(* Logix 5000 project; controller Arrow3 vendor 1 type 14 code 235 rev 36.11; software revision 36.00 *)

TASK MainTask (continuous, watchdog 500 ms) : MainProgram
TASK SafetyTask (periodic, rate 20 ms, priority 10, watchdog 20 ms, safety) : SafetyProgram

MODULES
   Local : vendor 1 type 14 code 235 (5069 0, rev 36.11)
      VRQx : vendor 1609 type 7 code 1234 (Ethernet 192.168.1.10, rev 1.4, StandardDataDriven RPI 20 ms)
END_MODULES

TYPE STR_20 :
STRUCT
   DATA : SINT[20];
END_STRUCT
END_TYPE

PROGRAM MainProgram   (* main routine MainRoutine *)
VAR
   b : BOOL := 1;
   DI1_4_INPUTTYPE_GET : MESSAGE;
        MessageParameters(ServiceCode := 16#000e, DestinationTag := DI1_4_INPUTTYPE_GET_VAL, ...)
   DI1_4_INPUTTYPE_GET_VAL : UINT;
   DI1_4_INPUTTYPE_SET : MESSAGE;
        MessageParameters(ServiceCode := 16#0010, LocalElement := DI1_4_INPUTTYPE_SET_VAL, ...)
   DI1_4_INPUTTYPE_SET_VAL : UINT;
   DI1_4_INPUTTYPE_TRG_GET : BOOL;
   DI1_4_INPUTTYPE_TRG_SET : BOOL;
   DI1_8_FORCEENABLE_GET : MESSAGE;
        MessageParameters(ServiceCode := 16#000e, DestinationTag := DI1_8_FORCEENABLE_GET_VAL, ...)
   DI1_8_FORCEENABLE_GET_VAL : UINT;
   DI1_8_FORCEENABLE_SET : MESSAGE;
        MessageParameters(ServiceCode := 16#0010, LocalElement := DI1_8_FORCEENABLE_SET_VAL, ...)
   DI1_8_FORCEENABLE_SET_VAL : UINT;
   DI1_8_FORCEENABLE_TRG_GET : BOOL;
   DI1_8_FORCEENABLE_TRG_SET : BOOL;
   DI1_8_FORCESTATE_GET : MESSAGE;
        MessageParameters(ServiceCode := 16#000e, DestinationTag := DI1_8_FORCESTATE_GET_VAL, ...)
   DI1_8_FORCESTATE_GET_VAL : UINT;
   DI1_8_FORCESTATE_SET : MESSAGE;
        MessageParameters(ServiceCode := 16#0010, LocalElement := DI1_8_FORCESTATE_SET_VAL, ...)
   DI1_8_FORCESTATE_SET_VAL : UINT;
   DI1_8_FORCESTATE_TRG_GET : BOOL;
   DI1_8_FORCESTATE_TRG_SET : BOOL;
   DI1_8_LOGICINVERT_GET : MESSAGE;
        MessageParameters(ServiceCode := 16#000e, DestinationTag := DI1_8_LOGICINVERT_GET_VAL, ...)
   DI1_8_LOGICINVERT_GET_VAL : UINT;
   DI1_8_LOGICINVERT_SET : MESSAGE;
        MessageParameters(ServiceCode := 16#0010, LocalElement := DI1_8_LOGICINVERT_SET_VAL, ...)
   DI1_8_LOGICINVERT_SET_VAL : UINT;
   DI1_8_LOGICINVERT_TRG_GET : BOOL;
   DI1_8_LOGICINVERT_TRG_SET : BOOL;
   DI1_CHNLERRSTS_GET : MESSAGE;
        MessageParameters(ServiceCode := 16#000e, DestinationTag := DI1_CHNLERRSTS_GET_VAL, ...)
   DI1_CHNLERRSTS_GET_VAL : UINT;
   DI1_CHNLERRSTS_TRG_GET : BOOL;
   DI1_DEBOUNCEDUR_GET : MESSAGE;
        MessageParameters(ServiceCode := 16#000e, DestinationTag := DI1_DEBOUNCEDUR_GET_VAL, ...)
   DI1_DEBOUNCEDUR_GET_VAL : UINT;
   DI1_DEBOUNCEDUR_SET : MESSAGE;
        MessageParameters(ServiceCode := 16#0010, LocalElement := DI1_DEBOUNCEDUR_SET_VAL, ...)
   DI1_DEBOUNCEDUR_SET_VAL : UINT;
   DI1_DEBOUNCEDUR_TRG_GET : BOOL := 1;
   DI1_DEBOUNCEDUR_TRG_SET : BOOL;
   DI1_HOLDDUR_SET : MESSAGE;
        MessageParameters(ServiceCode := 16#0010, LocalElement := DI1_HOLDDUR_SET_VAL, ...)
   DI1_HOLDDUR_SET_VAL : UINT;
   DI1_HOLDDUR_TRG_SET : BOOL;
   DI2_CHNLERRSTS_GET : MESSAGE;
        MessageParameters(ServiceCode := 16#000e, DestinationTag := DI2_CHNLERRSTS_GET_VAL, ...)
   DI2_CHNLERRSTS_GET_VAL : UINT;
   DI2_CHNLERRSTS_TRG_GET : BOOL;
   DI2_DEBOUNCEDUR_GET : MESSAGE;
        MessageParameters(ServiceCode := 16#000e, DestinationTag := DI2_DEBOUNCEDUR_GET_VAL, ...)
   DI2_DEBOUNCEDUR_GET_VAL : UINT;
   DI2_DEBOUNCEDUR_SET : MESSAGE;
        MessageParameters(ServiceCode := 16#0010, LocalElement := DI2_DEBOUNCEDUR_SET_VAL, ...)
   DI2_DEBOUNCEDUR_SET_VAL : UINT;
   DI2_DEBOUNCEDUR_TRG_GET : BOOL := 1;
   DI2_DEBOUNCEDUR_TRG_SET : BOOL;
   DI2_HOLDDUR_SET : MESSAGE;
        MessageParameters(ServiceCode := 16#0010, LocalElement := DI2_HOLDDUR_SET_VAL, ...)
   DI2_HOLDDUR_SET_VAL : UINT;
   DI2_HOLDDUR_TRG_SET : BOOL;
   DI3_CHNLERRSTS_GET : MESSAGE;
        MessageParameters(ServiceCode := 16#000e, DestinationTag := DI3_CHNLERRSTS_GET_VAL, ...)
   DI3_CHNLERRSTS_GET_VAL : UINT;
   DI3_CHNLERRSTS_TRG_GET : BOOL;
   DI3_DEBOUNCEDUR_GET : MESSAGE;
        MessageParameters(ServiceCode := 16#000e, DestinationTag := DI3_DEBOUNCEDUR_GET_VAL, ...)
   DI3_DEBOUNCEDUR_GET_VAL : UINT;
   DI3_DEBOUNCEDUR_SET : MESSAGE;
        MessageParameters(ServiceCode := 16#0010, LocalElement := DI3_DEBOUNCEDUR_SET_VAL, ...)
   DI3_DEBOUNCEDUR_SET_VAL : UINT;
   DI3_DEBOUNCEDUR_TRG_GET : BOOL := 1;
   DI3_DEBOUNCEDUR_TRG_SET : BOOL;
   DI3_HOLDDUR_SET : MESSAGE;
        MessageParameters(ServiceCode := 16#0010, LocalElement := DI3_HOLDDUR_SET_VAL, ...)
   DI3_HOLDDUR_SET_VAL : DINT;
   DI3_HOLDDUR_TRG_SET : BOOL;
   DI4_CHNLERRSTS_GET : MESSAGE;
        MessageParameters(ServiceCode := 16#000e, DestinationTag := DI4_CHNLERRSTS_GET_VAL, ...)
   DI4_CHNLERRSTS_GET_VAL : UINT;
   DI4_CHNLERRSTS_TRG_GET : BOOL;
   DI4_DEBOUNCEDUR_GET : MESSAGE;
        MessageParameters(ServiceCode := 16#000e, DestinationTag := DI4_DEBOUNCEDUR_GET_VAL, ...)
   DI4_DEBOUNCEDUR_GET_VAL : UINT;
   DI4_DEBOUNCEDUR_SET : MESSAGE;
        MessageParameters(ServiceCode := 16#0010, LocalElement := DI4_DEBOUNCEDUR_SET_VAL, ...)
   DI4_DEBOUNCEDUR_SET_VAL : UINT;
   DI4_DEBOUNCEDUR_TRG_GET : BOOL := 1;
   DI4_DEBOUNCEDUR_TRG_SET : BOOL;
   DI4_HOLDDUR_SET : MESSAGE;
        MessageParameters(ServiceCode := 16#0010, LocalElement := DI4_HOLDDUR_SET_VAL, ...)
   DI4_HOLDDUR_SET_VAL : UINT;
   DI4_HOLDDUR_TRG_SET : BOOL;
   DI5_8_INPUTTYPE_GET : MESSAGE;
        MessageParameters(ServiceCode := 16#000e, DestinationTag := DI5_8_INPUTTYPE_GET_VAL, ...)
   DI5_8_INPUTTYPE_GET_VAL : UINT;
   DI5_8_INPUTTYPE_SET : MESSAGE;
        MessageParameters(ServiceCode := 16#0010, LocalElement := DI5_8_INPUTTYPE_SET_VAL, ...)
   DI5_8_INPUTTYPE_SET_VAL : UINT;
   DI5_8_INPUTTYPE_TRG_GET : BOOL;
   DI5_8_INPUTTYPE_TRG_SET : BOOL;
   DI5_CHNLERRSTS_GET : MESSAGE;
        MessageParameters(ServiceCode := 16#000e, DestinationTag := DI5_CHNLERRSTS_GET_VAL, ...)
   DI5_CHNLERRSTS_GET_VAL : UINT;
   DI5_CHNLERRSTS_TRG_GET : BOOL;
   DI5_DEBOUNCEDUR_GET : MESSAGE;
        MessageParameters(ServiceCode := 16#000e, DestinationTag := DI5_DEBOUNCEDUR_GET_VAL, ...)
   DI5_DEBOUNCEDUR_GET_VAL : UINT;
   DI5_DEBOUNCEDUR_SET : MESSAGE;
        MessageParameters(ServiceCode := 16#0010, LocalElement := DI5_DEBOUNCEDUR_SET_VAL, ...)
   DI5_DEBOUNCEDUR_SET_VAL : UINT;
   DI5_DEBOUNCEDUR_TRG_GET : BOOL;
   DI5_DEBOUNCEDUR_TRG_SET : BOOL;
   DI5_HOLDDUR_SET : MESSAGE;
        MessageParameters(ServiceCode := 16#0010, LocalElement := DI5_HOLDDUR_SET_VAL, ...)
   DI5_HOLDDUR_SET_VAL : UINT;
   DI5_HOLDDUR_TRG_SET : BOOL;
   DI6_CHNLERRSTS_GET : MESSAGE;
        MessageParameters(ServiceCode := 16#000e, DestinationTag := DI6_CHNLERRSTS_GET_VAL, ...)
   DI6_CHNLERRSTS_GET_VAL : UINT;
   DI6_CHNLERRSTS_TRG_GET : BOOL;
   DI6_DEBOUNCEDUR_GET : MESSAGE;
        MessageParameters(ServiceCode := 16#000e, DestinationTag := DI6_DEBOUNCEDUR_GET_VAL, ...)
   DI6_DEBOUNCEDUR_GET_VAL : UINT;
   DI6_DEBOUNCEDUR_SET : MESSAGE;
        MessageParameters(ServiceCode := 16#0010, LocalElement := DI6_DEBOUNCEDUR_SET_VAL, ...)
   DI6_DEBOUNCEDUR_SET_VAL : UINT;
   DI6_DEBOUNCEDUR_TRG_GET : BOOL;
   DI6_DEBOUNCEDUR_TRG_SET : BOOL;
   DI6_HOLDDUR_SET : MESSAGE;
        MessageParameters(ServiceCode := 16#0010, LocalElement := DI6_HOLDDUR_SET_VAL, ...)
   DI6_HOLDDUR_SET_VAL : UINT;
   DI6_HOLDDUR_TRG_SET : BOOL;
   DI7_CHNLERRSTS_GET : MESSAGE;
        MessageParameters(ServiceCode := 16#000e, DestinationTag := DI7_CHNLERRSTS_GET_VAL, ...)
   DI7_CHNLERRSTS_GET_VAL : UINT;
   DI7_CHNLERRSTS_TRG_GET : BOOL;
   DI7_DEBOUNCEDUR_GET : MESSAGE;
        MessageParameters(ServiceCode := 16#000e, DestinationTag := DI7_DEBOUNCEDUR_GET_VAL, ...)
   DI7_DEBOUNCEDUR_GET_VAL : UINT;
   DI7_DEBOUNCEDUR_SET : MESSAGE;
        MessageParameters(ServiceCode := 16#0010, LocalElement := DI7_DEBOUNCEDUR_SET_VAL, ...)
   DI7_DEBOUNCEDUR_SET_VAL : UINT;
   DI7_DEBOUNCEDUR_TRG_GET : BOOL;
   DI7_DEBOUNCEDUR_TRG_SET : BOOL;
   DI7_HOLDDUR_SET : MESSAGE;
        MessageParameters(ServiceCode := 16#0010, LocalElement := DI7_HOLDDUR_SET_VAL, ...)
   DI7_HOLDDUR_SET_VAL : UINT;
   DI7_HOLDDUR_TRG_SET : BOOL;
   DI8_CHNLERRSTS_GET : MESSAGE;
        MessageParameters(ServiceCode := 16#000e, DestinationTag := DI8_CHNLERRSTS_GET_VAL, ...)
   DI8_CHNLERRSTS_GET_VAL : UINT;
   DI8_CHNLERRSTS_TRG_GET : BOOL;
   DI8_DEBOUNCEDUR_GET : MESSAGE;
        MessageParameters(ServiceCode := 16#000e, DestinationTag := DI8_DEBOUNCEDUR_GET_VAL, ...)
   DI8_DEBOUNCEDUR_GET_VAL : UINT;
   DI8_DEBOUNCEDUR_SET : MESSAGE;
        MessageParameters(ServiceCode := 16#0010, LocalElement := DI7_DEBOUNCEDUR_SET_VAL, ...)
   DI8_DEBOUNCEDUR_SET_VAL : UINT;
   DI8_DEBOUNCEDUR_TRG_GET : BOOL;
   DI8_DEBOUNCEDUR_TRG_SET : BOOL;
   DI8_HOLDDUR_SET : MESSAGE;
        MessageParameters(ServiceCode := 16#0010, LocalElement := DI8_HOLDDUR_SET_VAL, ...)
   DI8_HOLDDUR_SET_VAL : UINT;
   DI8_HOLDDUR_TRG_SET : BOOL;
   DI_BOTHEDGE_INT_GET : MESSAGE;
        MessageParameters(ServiceCode := 16#000e, DestinationTag := DI_BOTHEDGE_INT_GET_VAL, ...)
   DI_BOTHEDGE_INT_GET_VAL : UINT;
   DI_BOTHEDGE_INT_SET : MESSAGE;
        MessageParameters(ServiceCode := 16#0010, LocalElement := DI_BOTHEDGE_INT_SET_VAL, ...)
   DI_BOTHEDGE_INT_SET_VAL : DINT;
   DI_BOTHEDGE_INT_TRG_GET : BOOL;
   DI_BOTHEDGE_INT_TRG_SET : BOOL;
   DI_HITOLOEDGE_INT_GET : MESSAGE;
        MessageParameters(ServiceCode := 16#000e, DestinationTag := DI_HITOLOEDGE_INT_GET_VAL, ...)
   DI_HITOLOEDGE_INT_GET_VAL : UINT;
   DI_HITOLOEDGE_INT_SET : MESSAGE;
        MessageParameters(ServiceCode := 16#0010, LocalElement := DI_HITOLOEDGE_INT_SET_VAL, ...)
   DI_HITOLOEDGE_INT_SET_VAL : DINT;
   DI_HITOLOEDGE_INT_TRG_GET : BOOL;
   DI_HITOLOEDGE_INT_TRG_SET : BOOL;
   DI_LOTOHIEDGE_INT_GET : MESSAGE;
        MessageParameters(ServiceCode := 16#000e, DestinationTag := DI_LOTOHIEDGE_INT_GET_VAL, ...)
   DI_LOTOHIEDGE_INT_GET_VAL : UINT;
   DI_LOTOHIEDGE_INT_SET : MESSAGE;
        MessageParameters(ServiceCode := 16#0010, LocalElement := DI_LOTOHIEDGE_INT_SET_VAL, ...)
   DI_LOTOHIEDGE_INT_SET_VAL : DINT;
   DI_LOTOHIEDGE_INT_TRG_GET : BOOL;
   DI_LOTOHIEDGE_INT_TRG_SET : BOOL;
   DIO_CHNLPOS_ERRSTATUS_GET : MESSAGE;
        MessageParameters(ServiceCode := 16#000e, DestinationTag := DIO_CHNLPOS_ERRSTATUS_GET_VAL, ...)
   DIO_CHNLPOS_ERRSTATUS_GET_VAL : UINT;
   DIO_CHNLPOS_ERRSTATUS_TRG_GET : BOOL;
   DIO_FAULTRECOVERYENABLE_GET : MESSAGE;
        MessageParameters(ServiceCode := 16#000e, DestinationTag := DIO_FAULTRECOVERYENABLE_GET_VAL, ...)
   DIO_FAULTRECOVERYENABLE_GET_VAL : UINT;
   DIO_FAULTRECOVERYENABLE_SET : MESSAGE;
        MessageParameters(ServiceCode := 16#0010, LocalElement := DIO_FAULTRECOVERYENABLE_SET_VAL, ...)
   DIO_FAULTRECOVERYENABLE_SET_VAL : UINT;
   DIO_FAULTRECOVERYENABLE_TRG_GET : BOOL;
   DIO_FAULTRECOVERYENABLE_TRG_SET : BOOL;
   DIO_IDENT_DEVICEID_GET : MESSAGE;
        MessageParameters(ServiceCode := 16#000e, DestinationTag := DIO_IDENT_DEVICEID_GET_VAL, ...)
   DIO_IDENT_DEVICEID_GET_VAL : UDINT;
   DIO_IDENT_DEVICEID_TRG_GET : BOOL;
   DIO_IDENT_DEVICENAME_GET : MESSAGE;
        MessageParameters(ServiceCode := 16#000e, DestinationTag := DIO_IDENT_DEVICENAME_GET_VAL, ...)
   DIO_IDENT_DEVICENAME_GET_VAL : STR_20;
   DIO_IDENT_DEVICENAME_TRG_GET : BOOL;
   DIO_IDENT_DEVICETYPE_GET : MESSAGE;
        MessageParameters(ServiceCode := 16#000e, DestinationTag := DIO_IDENT_DEVICETYPE_GET_VAL, ...)
   DIO_IDENT_DEVICETYPE_GET_VAL : UDINT;
   DIO_IDENT_DEVICETYPE_TRG_GET : BOOL;
   DIO_IDENT_HWREV_GET : MESSAGE;
        MessageParameters(ServiceCode := 16#000e, DestinationTag := DIO_IDENT_HWREV_GET_VAL, ...)
   DIO_IDENT_HWREV_GET_VAL : STR_20;
   DIO_IDENT_HWREV_TRG_GET : BOOL;
   DIO_IDENT_SERIALNO_GET : MESSAGE;
        MessageParameters(ServiceCode := 16#000e, DestinationTag := DIO_IDENT_SERIALNO_GET_VAL, ...)
   DIO_IDENT_SERIALNO_GET_VAL : STR_20;
   DIO_IDENT_SERIALNO_TRG_GET : BOOL;
   DIO_IDENT_SWPARTNO_GET : MESSAGE;
        MessageParameters(ServiceCode := 16#000e, DestinationTag := DIO_IDENT_SWPARTNO_GET_VAL, ...)
   DIO_IDENT_SWPARTNO_GET_VAL : STR_20;
   DIO_IDENT_SWPARTNO_TRG_GET : BOOL;
   DIO_IDENT_SWREV_GET : MESSAGE;
        MessageParameters(ServiceCode := 16#000e, DestinationTag := DIO_IDENT_SWREV_GET_VAL, ...)
   DIO_IDENT_SWREV_GET_VAL : STR_20;
   DIO_IDENT_SWREV_TRG_GET : BOOL;
   DIO_IDENT_VARIANTID_GET : MESSAGE;
        MessageParameters(ServiceCode := 16#000e, DestinationTag := DIO_IDENT_VARIANTID_GET_VAL, ...)
   DIO_IDENT_VARIANTID_GET_VAL : STR_20;
   DIO_IDENT_VARIANTID_TRG_GET : BOOL;
   DIO_IDENT_VENDORID_GET : MESSAGE;
        MessageParameters(ServiceCode := 16#000e, DestinationTag := DIO_IDENT_VENDORID_GET_VAL, ...)
   DIO_IDENT_VENDORID_GET_VAL : UDINT;
   DIO_IDENT_VENDORID_TRG_GET : BOOL;
   DIO_IDENT_VENDORNAME_GET : MESSAGE;
        MessageParameters(ServiceCode := 16#000e, DestinationTag := DIO_IDENT_VENDORNAME_GET_VAL, ...)
   DIO_IDENT_VENDORNAME_GET_VAL : STR_20;
   DIO_IDENT_VENDORNAME_TRG_GET : BOOL;
   DIO_MEMORYLIFECYCLE_GET : MESSAGE;
        MessageParameters(ServiceCode := 16#000e, DestinationTag := DIO_MEMORYLIFECYCLE_GET_VAL, ...)
   DIO_MEMORYLIFECYCLE_GET_VAL : UDINT;
   DIO_MEMORYLIFECYCLE_TRG_GET : BOOL;
   DIO_OPERATIONTIME_HR_GET : MESSAGE;
        MessageParameters(ServiceCode := 16#000e, DestinationTag := DIO_OPERATIONTIME_HR_GET_VAL, ...)
   DIO_OPERATIONTIME_HR_GET_VAL : UDINT;
   DIO_OPERATIONTIME_HR_TRG_GET : BOOL;
   DIO_OPERATIONTIME_MIN_GET : MESSAGE;
        MessageParameters(ServiceCode := 16#000e, DestinationTag := DIO_OPERATIONTIME_MIN_GET_VAL, ...)
   DIO_OPERATIONTIME_MIN_GET_VAL : UDINT;
   DIO_OPERATIONTIME_MIN_TRG_GET : BOOL;
   DO1_8_BUSFAULTENABLE_GET : MESSAGE;
        MessageParameters(ServiceCode := 16#000e, DestinationTag := DO1_8_BUSFAULTENABLE_GET_VAL, ...)
   DO1_8_BUSFAULTENABLE_GET_VAL : UINT;
   DO1_8_BUSFAULTENABLE_SET : MESSAGE;
        MessageParameters(ServiceCode := 16#0010, LocalElement := DO1_8_BUSFAULTENABLE_SET_VAL, ...)
   DO1_8_BUSFAULTENABLE_SET_VAL : UINT;
   DO1_8_BUSFAULTENABLE_TRG_GET : BOOL;
   DO1_8_BUSFAULTENABLE_TRG_SET : BOOL;
   DO1_8_BUSFAULTSTATE_GET : MESSAGE;
        MessageParameters(ServiceCode := 16#000e, DestinationTag := DO1_8_BUSFAULTSTATE_GET_VAL, ...)
   DO1_8_BUSFAULTSTATE_GET_VAL : UINT;
   DO1_8_BUSFAULTSTATE_SET : MESSAGE;
        MessageParameters(ServiceCode := 16#0010, LocalElement := DO1_8_BUSFAULTSTATE_SET_VAL, ...)
   DO1_8_BUSFAULTSTATE_SET_VAL : UINT;
   DO1_8_BUSFAULTSTATE_TRG_GET : BOOL;
   DO1_8_BUSFAULTSTATE_TRG_SET : BOOL;
   DO1_8_FORCEENABLE_GET : MESSAGE;
        MessageParameters(ServiceCode := 16#000e, DestinationTag := DO1_8_FORCEENABLE_GET_VAL, ...)
   DO1_8_FORCEENABLE_GET_VAL : UINT;
   DO1_8_FORCEENABLE_SET : MESSAGE;
        MessageParameters(ServiceCode := 16#0010, LocalElement := DO1_8_FORCEENABLE_SET_VAL, ...)
   DO1_8_FORCEENABLE_SET_VAL : UINT;
   DO1_8_FORCEENABLE_TRG_GET : BOOL;
   DO1_8_FORCEENABLE_TRG_SET : BOOL;
   DO1_8_FORCESTATE_GET : MESSAGE;
        MessageParameters(ServiceCode := 16#000e, DestinationTag := DO1_8_FORCESTATE_GET_VAL, ...)
   DO1_8_FORCESTATE_GET_VAL : UINT;
   DO1_8_FORCESTATE_SET : MESSAGE;
        MessageParameters(ServiceCode := 16#0010, LocalElement := DO1_8_FORCESTATE_SET_VAL, ...)
   DO1_8_FORCESTATE_SET_VAL : UINT;
   DO1_8_FORCESTATE_TRG_GET : BOOL;
   DO1_8_FORCESTATE_TRG_SET : BOOL;
   DO1_8_IDLEMODEENABLE_GET : MESSAGE;
        MessageParameters(ServiceCode := 16#000e, DestinationTag := DO1_8_IDLEMODEENABLE_GET_VAL, ...)
   DO1_8_IDLEMODEENABLE_GET_VAL : UINT;
   DO1_8_IDLEMODEENABLE_SET : MESSAGE;
        MessageParameters(ServiceCode := 16#0010, LocalElement := DO1_8_IDLEMODEENABLE_SET_VAL, ...)
   DO1_8_IDLEMODEENABLE_SET_VAL : UINT;
   DO1_8_IDLEMODEENABLE_TRG_GET : BOOL;
   DO1_8_IDLEMODEENABLE_TRG_SET : BOOL;
   DO1_8_IDLEMODESTATE_GET : MESSAGE;
        MessageParameters(ServiceCode := 16#000e, DestinationTag := DO1_8_IDLEMODESTATE_GET_VAL, ...)
   DO1_8_IDLEMODESTATE_GET_VAL : UINT;
   DO1_8_IDLEMODESTATE_SET : MESSAGE;
        MessageParameters(ServiceCode := 16#0010, LocalElement := DO1_8_IDLEMODESTATE_SET_VAL, ...)
   DO1_8_IDLEMODESTATE_SET_VAL : UINT;
   DO1_8_IDLEMODESTATE_TRG_GET : BOOL;
   DO1_8_IDLEMODESTATE_TRG_SET : BOOL;
   DO1_CHNLERRSTS_GET : MESSAGE;
        MessageParameters(ServiceCode := 16#000e, DestinationTag := DO1_CHNLERRSTS_GET_VAL, ...)
   DO1_CHNLERRSTS_GET_VAL : UINT;
   DO1_CHNLERRSTS_TRG_GET : BOOL;
   DO2_CHNLERRSTS_GET : MESSAGE;
        MessageParameters(ServiceCode := 16#000e, DestinationTag := DO2_CHNLERRSTS_GET_VAL, ...)
   DO2_CHNLERRSTS_GET_VAL : UINT;
   DO2_CHNLERRSTS_TRG_GET : BOOL;
   DO3_CHNLERRSTS_GET : MESSAGE;
        MessageParameters(ServiceCode := 16#000e, DestinationTag := DO3_CHNLERRSTS_GET_VAL, ...)
   DO3_CHNLERRSTS_GET_VAL : UINT;
   DO3_CHNLERRSTS_TRG_GET : BOOL;
   DO4_CHNLERRSTS_GET : MESSAGE;
        MessageParameters(ServiceCode := 16#000e, DestinationTag := DO4_CHNLERRSTS_GET_VAL, ...)
   DO4_CHNLERRSTS_GET_VAL : UINT;
   DO4_CHNLERRSTS_TRG_GET : BOOL;
   DO5_CHNLERRSTS_GET : MESSAGE;
        MessageParameters(ServiceCode := 16#000e, DestinationTag := DO5_CHNLERRSTS_GET_VAL, ...)
   DO5_CHNLERRSTS_GET_VAL : UINT;
   DO5_CHNLERRSTS_TRG_GET : BOOL;
   DO6_CHNLERRSTS_GET : MESSAGE;
        MessageParameters(ServiceCode := 16#000e, DestinationTag := DO6_CHNLERRSTS_GET_VAL, ...)
   DO6_CHNLERRSTS_GET_VAL : UINT;
   DO6_CHNLERRSTS_TRG_GET : BOOL;
   DO7_CHNLERRSTS_GET : MESSAGE;
        MessageParameters(ServiceCode := 16#000e, DestinationTag := DO7_CHNLERRSTS_GET_VAL, ...)
   DO7_CHNLERRSTS_GET_VAL : UINT;
   DO7_CHNLERRSTS_TRG_GET : BOOL;
   DO8_CHNLERRSTS_GET : MESSAGE;
        MessageParameters(ServiceCode := 16#000e, DestinationTag := DO8_CHNLERRSTS_GET_VAL, ...)
   DO8_CHNLERRSTS_GET_VAL : UINT;
   DO8_CHNLERRSTS_TRG_GET : BOOL;
   DO_IDLEMODEENABLE_GET : MESSAGE;
        MessageParameters(ServiceCode := 16#000e, DestinationTag := DO_IDLEMODEENABLE_GET_VAL, ...)
   DO_IDLEMODEENABLE_GET_VAL : UINT;
   DO_IDLEMODEENABLE_SET : MESSAGE;
        MessageParameters(ServiceCode := 16#0010, LocalElement := DO_IDLEMODEENABLE_SET_VAL, ...)
   DO_IDLEMODEENABLE_SET_VAL : UINT;
   DO_IDLEMODEENABLE_TRG_GET : BOOL;
   DO_IDLEMODEENABLE_TRG_SET : BOOL;
   ENABLE_IMPLICIT_SET : MESSAGE;
        MessageParameters(ServiceCode := 16#0010, LocalElement := ENABLE_IMPLICIT_SET_CMD_VAL, ...)
   ENABLE_IMPLICIT_SET_CMD_VAL : UINT;
   ENABLE_IMPLICIT_TRG_SET : BOOL;
   ISEM_BCKPLANE_IDENT_DEVICEID_GET : MESSAGE;
        MessageParameters(ServiceCode := 16#000e, DestinationTag := ISEM_BCKPLANE_IDENT_DEVICEID_GET_VAL, ...)
   ISEM_BCKPLANE_IDENT_DEVICEID_GET_VAL : UDINT;
   ISEM_BCKPLANE_IDENT_DEVICEID_TRG_GET : BOOL;
   ISEM_BCKPLANE_IDENT_DEVICENAME_GET : MESSAGE;
        MessageParameters(ServiceCode := 16#000e, DestinationTag := ISEM_BCKPLANE_IDENT_DEVICENAME_GET_VAL, ...)
   ISEM_BCKPLANE_IDENT_DEVICENAME_GET_VAL : STR_20;
   ISEM_BCKPLANE_IDENT_DEVICENAME_TRG_GET : BOOL;
   ISEM_BCKPLANE_IDENT_DEVICETYPE_GET : MESSAGE;
        MessageParameters(ServiceCode := 16#000e, DestinationTag := ISEM_BCKPLANE_IDENT_DEVICETYPE_GET_VAL, ...)
   ISEM_BCKPLANE_IDENT_DEVICETYPE_GET_VAL : UDINT;
   ISEM_BCKPLANE_IDENT_DEVICETYPE_TRG_GET : BOOL;
   ISEM_BCKPLANE_IDENT_HWREV_GET : MESSAGE;
        MessageParameters(ServiceCode := 16#000e, DestinationTag := ISEM_BCKPLANE_IDENT_HWREV_GET_VAL, ...)
   ISEM_BCKPLANE_IDENT_HWREV_GET_VAL : STR_20;
   ISEM_BCKPLANE_IDENT_HWREV_TRG_GET : BOOL;
   ISEM_BCKPLANE_IDENT_SERIALNO_GET : MESSAGE;
        MessageParameters(ServiceCode := 16#000e, DestinationTag := ISEM_BCKPLANE_IDENT_SERIALNO_GET_VAL, ...)
   ISEM_BCKPLANE_IDENT_SERIALNO_GET_VAL : STR_20;
   ISEM_BCKPLANE_IDENT_SERIALNO_TRG_GET : BOOL;
   ISEM_BCKPLANE_IDENT_SWPARTNO_GET : MESSAGE;
        MessageParameters(ServiceCode := 16#000e, DestinationTag := ISEM_BCKPLANE_IDENT_SWPARTNO_GET_VAL, ...)
   ISEM_BCKPLANE_IDENT_SWPARTNO_GET_VAL : STR_20;
   ISEM_BCKPLANE_IDENT_SWPARTNO_TRG_GET : BOOL;
   ISEM_BCKPLANE_IDENT_SWREV_GET : MESSAGE;
        MessageParameters(ServiceCode := 16#000e, DestinationTag := ISEM_BCKPLANE_IDENT_SWREV_GET_VAL, ...)
   ISEM_BCKPLANE_IDENT_SWREV_GET_VAL : STR_20;
   ISEM_BCKPLANE_IDENT_SWREV_TRG_GET : BOOL;
   ISEM_BCKPLANE_IDENT_VARIANTID_GET : MESSAGE;
        MessageParameters(ServiceCode := 16#000e, DestinationTag := ISEM_BCKPLANE_IDENT_VARIANTID_GET_VAL, ...)
   ISEM_BCKPLANE_IDENT_VARIANTID_GET_VAL : STR_20;
   ISEM_BCKPLANE_IDENT_VARIANTID_TRG_GET : BOOL;
   ISEM_BCKPLANE_IDENT_VENDORID_GET : MESSAGE;
        MessageParameters(ServiceCode := 16#000e, DestinationTag := ISEM_BCKPLANE_IDENT_VENDORID_GET_VAL, ...)
   ISEM_BCKPLANE_IDENT_VENDORID_GET_VAL : UDINT;
   ISEM_BCKPLANE_IDENT_VENDORID_TRG_GET : BOOL;
   ISEM_BCKPLANE_IDENT_VENDORNAME_GET : MESSAGE;
        MessageParameters(ServiceCode := 16#000e, DestinationTag := ISEM_BCKPLANE_IDENT_VENDORNAME_GET_VAL, ...)
   ISEM_BCKPLANE_IDENT_VENDORNAME_GET_VAL : STR_20;
   ISEM_BCKPLANE_IDENT_VENDORNAME_TRG_GET : BOOL;
   ISEMDIAG_ApplPresHysteresis_GET : MESSAGE;
        MessageParameters(ServiceCode := 16#000e, DestinationTag := ISEMDIAG_ApplPresHysteresis_Get_VAL, ...)
   ISEMDIAG_ApplPresHysteresis_Get_VAL : INT;
   ISEMDIAG_ApplPresHysteresis_SET : MESSAGE;
        MessageParameters(ServiceCode := 16#0010, LocalElement := ISEMDIAG_ApplPresHysteresis_Set_VAL, ...)
   ISEMDIAG_ApplPresHysteresis_Set_VAL : INT;
   ISEMDIAG_ApplPresHysteresis_TRG_GET : BOOL;
   ISEMDIAG_ApplPresHysteresis_TRG_SET : BOOL;
   ISEMDIAG_FAULTEVNTBITS_GET : MESSAGE;
        MessageParameters(ServiceCode := 16#000e, DestinationTag := ISEMDIAG_FAULTEVNTBITS_GET_VAL, ...)
   ISEMDIAG_FAULTEVNTBITS_GET_VAL : UDINT;
   ISEMDIAG_FAULTEVNTBITS_TRG_GET : BOOL;
   ISEMDIAG_FAULTEVNTCOUNT_GET : MESSAGE;
        MessageParameters(ServiceCode := 16#000e, DestinationTag := ISEMDIAG_FAULTEVNTCOUNT_GET_VAL, ...)
   ISEMDIAG_FAULTEVNTCOUNT_GET_VAL : UINT;
   ISEMDIAG_FAULTEVNTCOUNT_TRG_GET : BOOL;
   ISEMDIAG_IDENT_DEVICEID_GET : MESSAGE;
        MessageParameters(ServiceCode := 16#000e, DestinationTag := ISEMDIAG_IDENT_DEVICEID_GET_VAL, ...)
   ISEMDIAG_IDENT_DEVICEID_GET_VAL : UDINT;
   ISEMDIAG_IDENT_DEVICEID_TRG_GET : BOOL;
   ISEMDIAG_IDENT_DEVICENAME_GET : MESSAGE;
        MessageParameters(ServiceCode := 16#000e, DestinationTag := ISEMDIAG_IDENT_DEVICENAME_GET_VAL, ...)
   ISEMDIAG_IDENT_DEVICENAME_GET_VAL : STR_20;
   ISEMDIAG_IDENT_DEVICENAME_TRG_GET : BOOL;
   ISEMDIAG_IDENT_DEVICETYPE_GET : MESSAGE;
        MessageParameters(ServiceCode := 16#000e, DestinationTag := ISEMDIAG_IDENT_DEVICETYPE_GET_VAL, ...)
   ISEMDIAG_IDENT_DEVICETYPE_GET_VAL : UDINT;
   ISEMDIAG_IDENT_DEVICETYPE_TRG_GET : BOOL;
   ISEMDIAG_IDENT_HWREV_GET : MESSAGE;
        MessageParameters(ServiceCode := 16#000e, DestinationTag := ISEMDIAG_IDENT_HWREV_GET_VAL, ...)
   ISEMDIAG_IDENT_HWREV_GET_VAL : STR_20;
   ISEMDIAG_IDENT_HWREV_TRG_GET : BOOL;
   ISEMDIAG_IDENT_SERIALNO_GET : MESSAGE;
        MessageParameters(ServiceCode := 16#000e, DestinationTag := ISEMDIAG_IDENT_SERIALNO_GET_VAL, ...)
   ISEMDIAG_IDENT_SERIALNO_GET_VAL : STR_20;
   ISEMDIAG_IDENT_SERIALNO_TRG_GET : BOOL;
   ISEMDIAG_IDENT_SWPARTNO_GET : MESSAGE;
        MessageParameters(ServiceCode := 16#000e, DestinationTag := ISEMDIAG_IDENT_SWPARTNO_GET_VAL, ...)
   ISEMDIAG_IDENT_SWPARTNO_GET_VAL : STR_20;
   ISEMDIAG_IDENT_SWPARTNO_TRG_GET : BOOL;
   ISEMDIAG_IDENT_SWREV_GET : MESSAGE;
        MessageParameters(ServiceCode := 16#000e, DestinationTag := ISEMDIAG_IDENT_SWREV_GET_VAL, ...)
   ISEMDIAG_IDENT_SWREV_GET_VAL : STR_20;
   ISEMDIAG_IDENT_SWREV_TRG_GET : BOOL;
   ISEMDIAG_IDENT_VARIANTID_GET : MESSAGE;
        MessageParameters(ServiceCode := 16#000e, DestinationTag := ISEMDIAG_IDENT_VARIANTID_GET_VAL, ...)
   ISEMDIAG_IDENT_VARIANTID_GET_VAL : STR_20;
   ISEMDIAG_IDENT_VARIANTID_TRG_GET : BOOL;
   ISEMDIAG_IDENT_VENDORID_GET : MESSAGE;
        MessageParameters(ServiceCode := 16#000e, DestinationTag := ISEMDIAG_IDENT_VENDORID_GET_VAL, ...)
   ISEMDIAG_IDENT_VENDORID_GET_VAL : UDINT;
   ISEMDIAG_IDENT_VENDORID_TRG_GET : BOOL;
   ISEMDIAG_IDENT_VENDORNAME_GET : MESSAGE;
        MessageParameters(ServiceCode := 16#000e, DestinationTag := ISEMDIAG_IDENT_VENDORNAME_GET_VAL, ...)
   ISEMDIAG_IDENT_VENDORNAME_GET_VAL : STR_20;
   ISEMDIAG_IDENT_VENDORNAME_TRG_GET : BOOL;
   ISEMDIAG_MaxApplPressure_GET : MESSAGE;
        MessageParameters(ServiceCode := 16#000e, DestinationTag := ISEMDIAG_MaxApplPressure_Get_VAL, ...)
   ISEMDIAG_MaxApplPressure_Get_VAL : INT;
   ISEMDIAG_MaxApplPressure_SET : MESSAGE;
        MessageParameters(ServiceCode := 16#0010, LocalElement := ISEMDIAG_MaxApplPressure_Set_VAL, ...)
   ISEMDIAG_MaxApplPressure_Set_VAL : INT;
   ISEMDIAG_MaxApplPressure_TRG_GET : BOOL;
   ISEMDIAG_MaxApplPressure_TRG_SET : BOOL;
   ISEMDIAG_MeasuredAuxCur_GET : MESSAGE;
        MessageParameters(ServiceCode := 16#000e, DestinationTag := ISEMDIAG_MeasuredAuxCur_GET_VAL, ...)
   ISEMDIAG_MeasuredAuxCur_GET_VAL : INT;
   ISEMDIAG_MeasuredAuxCur_TRG_GET : BOOL;
   ISEMDIAG_MeasuredAuxVolt_GET : MESSAGE;
        MessageParameters(ServiceCode := 16#000e, DestinationTag := ISEMDIAG_MeasuredAuxVolt_GET_VAL, ...)
   ISEMDIAG_MeasuredAuxVolt_GET_VAL : INT;
   ISEMDIAG_MeasuredAuxVolt_TRG_GET : BOOL;
   ISEMDIAG_MeasuredPressure_GET : MESSAGE;
        MessageParameters(ServiceCode := 16#000e, DestinationTag := ISEMDIAG_MeasuredPressure_GET_VAL, ...)
   ISEMDIAG_MeasuredPressure_GET_VAL : INT;
   ISEMDIAG_MeasuredPressure_TRG_GET : BOOL;
   ISEMDIAG_MinApplPressure_GET : MESSAGE;
        MessageParameters(ServiceCode := 16#000e, DestinationTag := ISEMDIAG_MinApplPressure_Get_VAL, ...)
   ISEMDIAG_MinApplPressure_Get_VAL : INT;
   ISEMDIAG_MinApplPressure_SET : MESSAGE;
        MessageParameters(ServiceCode := 16#0010, LocalElement := ISEMDIAG_MinApplPressure_Set_VAL, ...)
   ISEMDIAG_MinApplPressure_Set_VAL : INT;
   ISEMDIAG_MinApplPressure_TRG_GET : BOOL;
   ISEMDIAG_MinApplPressure_TRG_SET : BOOL;
   ISEMDIAG_MinRatedPressure_GET : MESSAGE;
        MessageParameters(ServiceCode := 16#000e, DestinationTag := ISEMDIAG_MinRatedPressure_GET_VAL, ...)
   ISEMDIAG_MinRatedPressure_GET_VAL : DINT;
   ISEMDIAG_MinRatedPressure_TRG_GET : BOOL;
   ISEMDIAG_OPERATIONTIME_HR_GET : MESSAGE;
        MessageParameters(ServiceCode := 16#000e, DestinationTag := ISEMDIAG_OPERATIONTIME_HR_GET_VAL, ...)
   ISEMDIAG_OPERATIONTIME_HR_GET_VAL : UDINT;
   ISEMDIAG_OPERATIONTIME_HR_TRG_GET : BOOL;
   ISEMDIAG_OPERATIONTIME_MIN_GET : MESSAGE;
        MessageParameters(ServiceCode := 16#000e, DestinationTag := ISEMDIAG_OPERATIONTIME_MIN_GET_VAL, ...)
   ISEMDIAG_OPERATIONTIME_MIN_GET_VAL : UINT;
   ISEMDIAG_OPERATIONTIME_MIN_TRG_GET : BOOL;
   ISEMDIAG_POST_ERRSTS_GET : MESSAGE;
        MessageParameters(ServiceCode := 16#000e, DestinationTag := ISEMDIAG_POST_ERRSTS_GET_VAL, ...)
   ISEMDIAG_POST_ERRSTS_GET_VAL : UDINT;
   ISEMDIAG_POST_ERRSTS_TRG_GET : BOOL;
   ISEMDIAG_PWRONTIME_HR_GET : MESSAGE;
        MessageParameters(ServiceCode := 16#000e, DestinationTag := ISEMDIAG_PWRONTIME_HR_GET_VAL, ...)
   ISEMDIAG_PWRONTIME_HR_GET_VAL : UDINT;
   ISEMDIAG_PWRONTIME_HR_TRG_GET : BOOL;
   ISEMDIAG_PWRONTIME_MIN_GET : MESSAGE;
        MessageParameters(ServiceCode := 16#000e, DestinationTag := ISEMDIAG_PWRONTIME_MIN_GET_VAL, ...)
   ISEMDIAG_PWRONTIME_MIN_GET_VAL : UINT;
   ISEMDIAG_PWRONTIME_MIN_TRG_GET : BOOL;
   ISEMDIAG_RatedAuxCurHyst_GET : MESSAGE;
        MessageParameters(ServiceCode := 16#000e, DestinationTag := ISEMDIAG_RatedAuxCurHyst_Get_VAL, ...)
   ISEMDIAG_RatedAuxCurHyst_Get_VAL : INT;
   ISEMDIAG_RatedAuxCurHyst_SET : MESSAGE;
        MessageParameters(ServiceCode := 16#0010, LocalElement := ISEMDIAG_RatedAuxCurHyst_Set_VAL, ...)
   ISEMDIAG_RatedAuxCurHyst_Set_VAL : INT;
   ISEMDIAG_RatedAuxCurHyst_TRG_GET : BOOL;
   ISEMDIAG_RatedAuxCurHyst_TRG_SET : BOOL;
   ISEMDIAG_RatedAuxVoltHyst_GET : MESSAGE;
        MessageParameters(ServiceCode := 16#000e, DestinationTag := ISEMDIAG_RatedAuxVoltHyst_Get_VAL, ...)
   ISEMDIAG_RatedAuxVoltHyst_Get_VAL : INT;
   ISEMDIAG_RatedAuxVoltHyst_SET : MESSAGE;
        MessageParameters(ServiceCode := 16#0010, LocalElement := ISEMDIAG_RatedAuxVoltHyst_Set_VAL, ...)
   ISEMDIAG_RatedAuxVoltHyst_Set_VAL : INT;
   ISEMDIAG_RatedAuxVoltHyst_TRG_GET : BOOL;
   ISEMDIAG_RatedAuxVoltHyst_TRG_SET : BOOL;
   ISEMDIAG_WARNEVNTBITS_GET : MESSAGE;
        MessageParameters(ServiceCode := 16#000e, DestinationTag := ISEMDIAG_WARNEVNTBITS_GET_VAL, ...)
   ISEMDIAG_WARNEVNTBITS_GET_VAL : UDINT;
   ISEMDIAG_WARNEVNTBITS_TRG_GET : BOOL;
   ISEMDIAG_WARNEVNTCOUNT_GET : MESSAGE;
        MessageParameters(ServiceCode := 16#000e, DestinationTag := ISEMDIAG_WARNEVNTCOUNT_GET_VAL, ...)
   ISEMDIAG_WARNEVNTCOUNT_GET_VAL : UINT;
   ISEMDIAG_WARNEVNTCOUNT_TRG_GET : BOOL;
   ISEMDIAG_WARNSTSBITS_GET : MESSAGE;
        MessageParameters(ServiceCode := 16#000e, DestinationTag := ISEMDIAG_WARNSTSBITS_GET_VAL, ...)
   ISEMDIAG_WARNSTSBITS_GET_VAL : UDINT;
   ISEMDIAG_WARNSTSBITS_TRG_GET : BOOL;
   off_delay_timer : TIMER := (PRE := 100);
   on : BOOL := 1;
   On_Delay_Timer_1 : TIMER := (PRE := 100);
   On_Delay_Timer_10 : TIMER := (PRE := 500);
   On_Delay_Timer_11 : TIMER := (PRE := 550);
   On_Delay_Timer_12 : TIMER := (PRE := 600);
   On_Delay_Timer_13 : TIMER := (PRE := 650);
   On_Delay_Timer_14 : TIMER := (PRE := 700);
   On_Delay_Timer_15 : TIMER := (PRE := 750);
   On_Delay_Timer_16 : TIMER := (PRE := 800);
   On_Delay_Timer_2 : TIMER := (PRE := 200);
   On_Delay_Timer_3 : TIMER := (PRE := 300);
   On_Delay_Timer_4 : TIMER := (PRE := 400);
   On_Delay_Timer_5 : TIMER := (PRE := 500);
   On_Delay_Timer_6 : TIMER := (PRE := 600);
   On_Delay_Timer_7 : TIMER := (PRE := 700);
   On_Delay_Timer_8 : TIMER := (PRE := 800);
   On_Delay_Timer_9 : TIMER := (PRE := 450);
   on_delay_tmr : TIMER := (PRE := 800);
   POST_ERRSTS_GET : MESSAGE;
        MessageParameters(ServiceCode := 16#000e, DestinationTag := POST_ERRSTS_GET_VAL, ...)
   POST_ERRSTS_GET_VAL : UDINT;
   POST_ERRSTS_TRG_GET : BOOL;
   PROP_BCKPLANE_IDENT_DEVICEID_GET : MESSAGE;
        MessageParameters(ServiceCode := 16#000e, DestinationTag := PROP_BCKPLANE_IDENT_DEVICEID_GET_VAL, ...)
   PROP_BCKPLANE_IDENT_DEVICEID_GET_VAL : UDINT;
   PROP_BCKPLANE_IDENT_DEVICEID_TRG_GET : BOOL;
   PROP_BCKPLANE_IDENT_DEVICENAME_GET : MESSAGE;
        MessageParameters(ServiceCode := 16#000e, DestinationTag := PROP_BCKPLANE_IDENT_DEVICENAME_GET_VAL, ...)
   PROP_BCKPLANE_IDENT_DEVICENAME_GET_VAL : STR_20;
   PROP_BCKPLANE_IDENT_DEVICENAME_TRG_GET : BOOL;
   PROP_BCKPLANE_IDENT_DEVICETYPE_GET : MESSAGE;
        MessageParameters(ServiceCode := 16#000e, DestinationTag := PROP_BCKPLANE_IDENT_DEVICETYPE_GET_VAL, ...)
   PROP_BCKPLANE_IDENT_DEVICETYPE_GET_VAL : UDINT;
   PROP_BCKPLANE_IDENT_DEVICETYPE_TRG_GET : BOOL;
   PROP_BCKPLANE_IDENT_HWREV_GET : MESSAGE;
        MessageParameters(ServiceCode := 16#000e, DestinationTag := PROP_BCKPLANE_IDENT_HWREV_GET_VAL, ...)
   PROP_BCKPLANE_IDENT_HWREV_GET_VAL : STR_20;
   PROP_BCKPLANE_IDENT_HWREV_TRG_GET : BOOL;
   PROP_BCKPLANE_IDENT_SERIALNO_GET : MESSAGE;
        MessageParameters(ServiceCode := 16#000e, DestinationTag := PROP_BCKPLANE_IDENT_SERIALNO_GET_VAL, ...)
   PROP_BCKPLANE_IDENT_SERIALNO_GET_VAL : STR_20;
   PROP_BCKPLANE_IDENT_SERIALNO_TRG_GET : BOOL;
   PROP_BCKPLANE_IDENT_SWPARTNO_GET : MESSAGE;
        MessageParameters(ServiceCode := 16#000e, DestinationTag := PROP_BCKPLANE_IDENT_SWPARTNO_GET_VAL, ...)
   PROP_BCKPLANE_IDENT_SWPARTNO_GET_VAL : STR_20;
   PROP_BCKPLANE_IDENT_SWPARTNO_TRG_GET : BOOL;
   PROP_BCKPLANE_IDENT_SWREV_GET : MESSAGE;
        MessageParameters(ServiceCode := 16#000e, DestinationTag := PROP_BCKPLANE_IDENT_SWREV_GET_VAL, ...)
   PROP_BCKPLANE_IDENT_SWREV_GET_VAL : STR_20;
   PROP_BCKPLANE_IDENT_SWREV_TRG_GET : BOOL;
   PROP_BCKPLANE_IDENT_VARIANTID_GET : MESSAGE;
        MessageParameters(ServiceCode := 16#000e, DestinationTag := PROP_BCKPLANE_IDENT_VARIANTID_GET_VAL, ...)
   PROP_BCKPLANE_IDENT_VARIANTID_GET_VAL : STR_20;
   PROP_BCKPLANE_IDENT_VARIANTID_TRG_GET : BOOL;
   PROP_BCKPLANE_IDENT_VENDORID_GET : MESSAGE;
        MessageParameters(ServiceCode := 16#000e, DestinationTag := PROP_BCKPLANE_IDENT_VENDORID_GET_VAL, ...)
   PROP_BCKPLANE_IDENT_VENDORID_GET_VAL : UDINT;
   PROP_BCKPLANE_IDENT_VENDORID_TRG_GET : BOOL;
   PROP_BCKPLANE_IDENT_VENDORNAME_GET : MESSAGE;
        MessageParameters(ServiceCode := 16#000e, DestinationTag := PROP_BCKPLANE_IDENT_VENDORNAME_GET_VAL, ...)
   PROP_BCKPLANE_IDENT_VENDORNAME_GET_VAL : STR_20;
   PROP_BCKPLANE_IDENT_VENDORNAME_TRG_GET : BOOL;
   PROP_INTR_CONTROL_KD_GET : MESSAGE;
        MessageParameters(ServiceCode := 16#000e, DestinationTag := PROP_INTR_CONTROL_KD_Get_VAL, ...)
   PROP_INTR_CONTROL_KD_Get_VAL : UINT;
   PROP_INTR_CONTROL_KD_SET : MESSAGE;
        MessageParameters(ServiceCode := 16#0010, LocalElement := PROP_INTR_CONTROL_KD_set_VAL, ...)
   PROP_INTR_CONTROL_KD_set_VAL : UINT;
   PROP_INTR_CONTROL_KD_TRG_GET : BOOL;
   PROP_INTR_CONTROL_KD_TRG_SET : BOOL;
   PROP_INTR_CONTROL_KI_GET : MESSAGE;
        MessageParameters(ServiceCode := 16#000e, DestinationTag := PROP_INTR_CONTROL_KI_Get_VAL, ...)
   PROP_INTR_CONTROL_KI_Get_VAL : UINT;
   PROP_INTR_CONTROL_KI_SET : MESSAGE;
        MessageParameters(ServiceCode := 16#0010, LocalElement := PROP_INTR_CONTROL_KI_set_VAL, ...)
   PROP_INTR_CONTROL_KI_set_VAL : UINT;
   PROP_INTR_CONTROL_KI_TRG_GET : BOOL;
   PROP_INTR_CONTROL_KI_TRG_SET : BOOL;
   PROP_INTR_CONTROL_KP_GET : MESSAGE;
        MessageParameters(ServiceCode := 16#000e, DestinationTag := PROP_INTR_CONTROL_KP_Get_VAL, ...)
   PROP_INTR_CONTROL_KP_Get_VAL : UINT;
   PROP_INTR_CONTROL_KP_SET : MESSAGE;
        MessageParameters(ServiceCode := 16#0010, LocalElement := PROP_INTR_CONTROL_KP_Set_VAL, ...)
   PROP_INTR_CONTROL_KP_Set_VAL : UINT;
   PROP_INTR_CONTROL_KP_TRG_GET : BOOL;
   PROP_INTR_CONTROL_KP_TRG_SET : BOOL;
   PROP_INTR_CONTROL_LCDBRIGHT_GET : MESSAGE;
        MessageParameters(ServiceCode := 16#000e, DestinationTag := PROP_INTR_CONTROL_LCDBRIGHT_Get_VAL, ...)
   PROP_INTR_CONTROL_LCDBRIGHT_Get_VAL : UINT;
   PROP_INTR_CONTROL_LCDBRIGHT_SET : MESSAGE;
        MessageParameters(ServiceCode := 16#0010, LocalElement := PROP_INTR_CONTROL_LCDBRIGHT_Set_VAL, ...)
   PROP_INTR_CONTROL_LCDBRIGHT_Set_VAL : UINT;
   PROP_INTR_CONTROL_LCDBRIGHT_TRG_GET : BOOL;
   PROP_INTR_CONTROL_LCDBRIGHT_TRG_SET : BOOL;
   PROP_INTR_CONTROL_SPANADJST_GET : MESSAGE;
        MessageParameters(ServiceCode := 16#000e, DestinationTag := PROP_INTR_CONTROL_SPANADJST_Get_VAL, ...)
   PROP_INTR_CONTROL_SPANADJST_Get_VAL : INT;
   PROP_INTR_CONTROL_SPANADJST_SET : MESSAGE;
        MessageParameters(ServiceCode := 16#0010, LocalElement := PROP_INTR_CONTROL_SPANADJST_set_VAL, ...)
   PROP_INTR_CONTROL_SPANADJST_set_VAL : INT;
   PROP_INTR_CONTROL_SPANADJST_TRG_GET : BOOL;
   PROP_INTR_CONTROL_SPANADJST_TRG_SET : BOOL;
   PROP_INTR_CONTROL_ZEROADJST_GET : MESSAGE;
        MessageParameters(ServiceCode := 16#000e, DestinationTag := PROP_INTR_CONTROL_ZEROADJST_Get_VAL, ...)
   PROP_INTR_CONTROL_ZEROADJST_Get_VAL : INT;
   PROP_INTR_CONTROL_ZEROADJST_SET : MESSAGE;
        MessageParameters(ServiceCode := 16#0010, LocalElement := PROP_INTR_CONTROL_ZEROADJST_Set_VAL, ...)
   PROP_INTR_CONTROL_ZEROADJST_Set_VAL : INT;
   PROP_INTR_CONTROL_ZEROADJST_TRG_GET : BOOL;
   PROP_INTR_CONTROL_ZEROADJST_TRG_SET : BOOL;
   PROP_INTR_CYCLECOUNTER_GET : MESSAGE;
        MessageParameters(ServiceCode := 16#000e, DestinationTag := PROP_INTR_CYCLECOUNTER_GET_VAL, ...)
   PROP_INTR_CYCLECOUNTER_GET_VAL : UDINT;
   PROP_INTR_CYCLECOUNTER_TRG_GET : BOOL;
   PROP_INTR_IDENT_DEVICEID_GET : MESSAGE;
        MessageParameters(ServiceCode := 16#000e, DestinationTag := PROP_INTR_IDENT_DEVICEID_GET_VAL, ...)
   PROP_INTR_IDENT_DEVICEID_GET_VAL : UDINT;
   PROP_INTR_IDENT_DEVICEID_TRG_GET : BOOL;
   PROP_INTR_IDENT_DEVICENAME_GET : MESSAGE;
        MessageParameters(ServiceCode := 16#000e, DestinationTag := PROP_INTR_IDENT_DEVICENAME_GET_VAL, ...)
   PROP_INTR_IDENT_DEVICENAME_GET_VAL : STR_20;
   PROP_INTR_IDENT_DEVICENAME_TRG_GET : BOOL;
   PROP_INTR_IDENT_DEVICETYPE_GET : MESSAGE;
        MessageParameters(ServiceCode := 16#000e, DestinationTag := PROP_INTR_IDENT_DEVICETYPE_GET_VAL, ...)
   PROP_INTR_IDENT_DEVICETYPE_GET_VAL : UDINT;
   PROP_INTR_IDENT_DEVICETYPE_TRG_GET : BOOL;
   PROP_INTR_IDENT_HWREV_GET : MESSAGE;
        MessageParameters(ServiceCode := 16#000e, DestinationTag := PROP_INTR_IDENT_HWREV_GET_VAL, ...)
   PROP_INTR_IDENT_HWREV_GET_VAL : STR_20;
   PROP_INTR_IDENT_HWREV_TRG_GET : BOOL;
   PROP_INTR_IDENT_SERIALNO_GET : MESSAGE;
        MessageParameters(ServiceCode := 16#000e, DestinationTag := PROP_INTR_IDENT_SERIALNO_GET_VAL, ...)
   PROP_INTR_IDENT_SERIALNO_GET_VAL : STR_20;
   PROP_INTR_IDENT_SERIALNO_TRG_GET : BOOL;
   PROP_INTR_IDENT_SWPARTNO_GET : MESSAGE;
        MessageParameters(ServiceCode := 16#000e, DestinationTag := PROP_INTR_IDENT_SWPARTNO_GET_VAL, ...)
   PROP_INTR_IDENT_SWPARTNO_GET_VAL : STR_20;
   PROP_INTR_IDENT_SWPARTNO_TRG_GET : BOOL;
   PROP_INTR_IDENT_SWREV_GET : MESSAGE;
        MessageParameters(ServiceCode := 16#000e, DestinationTag := PROP_INTR_IDENT_SWREV_GET_VAL, ...)
   PROP_INTR_IDENT_SWREV_GET_VAL : STR_20;
   PROP_INTR_IDENT_SWREV_TRG_GET : BOOL;
   PROP_INTR_IDENT_VARIANTID_GET : MESSAGE;
        MessageParameters(ServiceCode := 16#000e, DestinationTag := PROP_INTR_IDENT_VARIANTID_GET_VAL, ...)
   PROP_INTR_IDENT_VARIANTID_GET_VAL : STR_20;
   PROP_INTR_IDENT_VARIANTID_TRG_GET : BOOL;
   PROP_INTR_IDENT_VENDORID_GET : MESSAGE;
        MessageParameters(ServiceCode := 16#000e, DestinationTag := PROP_INTR_IDENT_VENDORID_GET_VAL, ...)
   PROP_INTR_IDENT_VENDORID_GET_VAL : UDINT;
   PROP_INTR_IDENT_VENDORID_TRG_GET : BOOL;
   PROP_INTR_IDENT_VENDORNAME_GET : MESSAGE;
        MessageParameters(ServiceCode := 16#000e, DestinationTag := PROP_INTR_IDENT_VENDORNAME_GET_VAL, ...)
   PROP_INTR_IDENT_VENDORNAME_GET_VAL : STR_20;
   PROP_INTR_IDENT_VENDORNAME_TRG_GET : BOOL;
   PROP_INTR_OPRHR_GET : MESSAGE;
        MessageParameters(ServiceCode := 16#000e, DestinationTag := PROP_INTR_OPRHR_GET_VAL, ...)
   PROP_INTR_OPRHR_GET_VAL : UDINT;
   PROP_INTR_OPRHR_TRG_GET : BOOL;
   PROP_INTR_OPRMIN_GET : MESSAGE;
        MessageParameters(ServiceCode := 16#000e, DestinationTag := PROP_INTR_OPRMIN_GET_VAL, ...)
   PROP_INTR_OPRMIN_GET_VAL : UINT;
   PROP_INTR_OPRMIN_TRG_GET : BOOL;
   PROP_INTR_POST_ERRSTS_GET : MESSAGE;
        MessageParameters(ServiceCode := 16#000e, DestinationTag := PROP_INTR_POST_ERRSTS_GET_VAL, ...)
   PROP_INTR_POST_ERRSTS_GET_VAL : UDINT;
   PROP_INTR_POST_ERRSTS_TRG_GET : BOOL;
   PROP_INTR_TEMPERATURE_GET : MESSAGE;
        MessageParameters(ServiceCode := 16#000e, DestinationTag := PROP_INTR_TEMPERATURE_GET_VAL, ...)
   PROP_INTR_TEMPERATURE_GET_VAL : UINT;
   PROP_INTR_TEMPERATURE_TRG_GET : BOOL;
   PZ_DIAG_VALVE_POSITION_GET_VAL : UINT;
   PZ_DIAGVALVE_POSITION_GET : MESSAGE;
        MessageParameters(ServiceCode := 16#000e, DestinationTag := PZ_DIAG_VALVE_POSITION_GET_VAL, ...)
   PZ_DIAGVALVE_POSITION_TRG_GET : BOOL;
   PZ_ID_GET : MESSAGE;
        MessageParameters(ServiceCode := 16#000e, DestinationTag := PZ_ID_GET_VAL, ...)
   PZ_ID_GET_VAL : UINT;
   PZ_ID_TRG_GET : BOOL;
   PZ_IISEMDIAG_PRESENT_GET : MESSAGE;
        MessageParameters(ServiceCode := 16#000e, DestinationTag := PZ_ISEM_DIAG_PRESENT_GET_VAL, ...)
   PZ_IISEMDIAG_PRESENT_TRG_GET : BOOL;
   PZ_ISEM_DIAG_PRESENT_GET_VAL : UINT;
   PZ_NO_OF_STATIONS_GET_VAL : UINT;
   PZ_NOOFSTATIONS_GET : MESSAGE;
        MessageParameters(ServiceCode := 16#000e, DestinationTag := PZ_NO_OF_STATIONS_GET_VAL, ...)
   PZ_NOOFSTATIONS_TRG_GET : BOOL;
   PZ_PROP_EXTERNAL_PORT_GET : MESSAGE;
        MessageParameters(ServiceCode := 16#000e, DestinationTag := PZ_PROP_EXTERNAL_PORT_GET_VAL, ...)
   PZ_PROP_EXTERNAL_PORT_GET_VAL : UINT;
   PZ_PROP_EXTERNAL_PORT_TRG_GET : BOOL;
   SENSORSUPPLY_ENABLE_GET : MESSAGE;
        MessageParameters(ServiceCode := 16#000e, DestinationTag := SENSORSUPPLY_ENABLE_GET_VAL, ...)
   SENSORSUPPLY_ENABLE_GET_VAL : DINT;
   SENSORSUPPLY_ENABLE_SET : MESSAGE;
        MessageParameters(ServiceCode := 16#0010, LocalElement := SENSORSUPPLY_ENABLE_SET_VAL, ...)
   SENSORSUPPLY_ENABLE_SET_VAL : UINT;
   SENSORSUPPLY_ENABLE_TRG_GET : BOOL;
   SENSORSUPPLY_ENABLE_TRG_SET : BOOL;
   SENSUPL_SHRTCKTDIAGEN_GET : MESSAGE;
        MessageParameters(ServiceCode := 16#000e, DestinationTag := SENSUPL_SHRTCKTDIAGEN_GET_VAL, ...)
   SENSUPL_SHRTCKTDIAGEN_GET_VAL : DINT;
   SENSUPL_SHRTCKTDIAGEN_SET : MESSAGE;
        MessageParameters(ServiceCode := 16#0010, LocalElement := SENSUPL_SHRTCKTDIAGEN_SET_VAL, ...)
   SENSUPL_SHRTCKTDIAGEN_SET_VAL : UINT;
   SENSUPL_SHRTCKTDIAGEN_TRG_GET : BOOL;
   SENSUPL_SHRTCKTDIAGEN_TRG_SET : BOOL;
   STA_ApplPresHysteresis_GET : MESSAGE;
        MessageParameters(ServiceCode := 16#000e, DestinationTag := STA_ApplPresHysteresis_Get_VAL, ...)
   STA_ApplPresHysteresis_Get_VAL : INT;
   STA_ApplPresHysteresis_SET : MESSAGE;
        MessageParameters(ServiceCode := 16#0010, LocalElement := STA_ApplPresHysteresis_Set_VAL, ...)
   STA_ApplPresHysteresis_Set_VAL : INT;
   STA_ApplPresHysteresis_TRG_GET : BOOL;
   STA_ApplPresHysteresis_TRG_SET : BOOL;
   STA_Coil12HitCurHysteresis_GET : MESSAGE;
        MessageParameters(ServiceCode := 16#000e, DestinationTag := STA_Coil12HitCurHysteresis_Get_VAL, ...)
   STA_Coil12HitCurHysteresis_Get_VAL : INT;
   STA_Coil12HitCurHysteresis_SET : MESSAGE;
        MessageParameters(ServiceCode := 16#0010, LocalElement := STA_Coil12HitCurHysteresis_Set_VAL, ...)
   STA_Coil12HitCurHysteresis_Set_VAL : INT;
   STA_Coil12HitCurHysteresis_TRG_GET : BOOL;
   STA_Coil12HitCurHysteresis_TRG_SET : BOOL;
   STA_Coil12HitCurrent_GET : MESSAGE;
        MessageParameters(ServiceCode := 16#000e, DestinationTag := STA_Coil12HitCurrent_GET_VAL, ...)
   STA_Coil12HitCurrent_GET_VAL : INT;
   STA_Coil12HitCurrent_TRG_GET : BOOL;
   STA_Coil12HitPower_GET : MESSAGE;
        MessageParameters(ServiceCode := 16#000e, DestinationTag := STA_Coil12HitPower_GET_VAL, ...)
   STA_Coil12HitPower_GET_VAL : INT;
   STA_Coil12HitPower_TRG_GET : BOOL;
   STA_Coil12HoldCurrent_GET : MESSAGE;
        MessageParameters(ServiceCode := 16#000e, DestinationTag := STA_Coil12HoldCurrent_GET_VAL, ...)
   STA_Coil12HoldCurrent_GET_VAL : INT;
   STA_Coil12HoldCurrent_TRG_GET : BOOL;
   STA_Coil12HoldPower_GET : MESSAGE;
        MessageParameters(ServiceCode := 16#000e, DestinationTag := STA_Coil12HoldPower_Get_VAL, ...)
   STA_Coil12HoldPower_Get_VAL : INT;
   STA_Coil12HoldPower_SET : MESSAGE;
        MessageParameters(ServiceCode := 16#0010, LocalElement := STA_Coil12HoldPower_Set_VAL, ...)
   STA_Coil12HoldPower_Set_VAL : INT;
   STA_Coil12HoldPower_TRG_GET : BOOL;
   STA_Coil12HoldPower_TRG_SET : BOOL;
   STA_Coil12HoldVolage_GET : MESSAGE;
        MessageParameters(ServiceCode := 16#000e, DestinationTag := STA_Coil12HoldVolage_Get_VAL, ...)
   STA_Coil12HoldVolage_Get_VAL : INT;
   STA_Coil12HoldVolage_SET : MESSAGE;
        MessageParameters(ServiceCode := 16#0010, LocalElement := STA_Coil12HoldVolage_Set_VAL, ...)
   STA_Coil12HoldVolage_Set_VAL : INT;
   STA_Coil12HoldVolage_TRG_GET : BOOL;
   STA_Coil12HoldVolage_TRG_SET : BOOL;
   STA_Coil14HitCurHysteresis_GET : MESSAGE;
        MessageParameters(ServiceCode := 16#000e, DestinationTag := STA_Coil14HitCurHysteresis_Get_VAL, ...)
   STA_Coil14HitCurHysteresis_Get_VAL : INT;
   STA_Coil14HitCurHysteresis_SET : MESSAGE;
        MessageParameters(ServiceCode := 16#0010, LocalElement := STA_Coil14HitCurHysteresis_Set_VAL, ...)
   STA_Coil14HitCurHysteresis_Set_VAL : INT;
   STA_Coil14HitCurHysteresis_TRG_GET : BOOL;
   STA_Coil14HitCurHysteresis_TRG_SET : BOOL;
   STA_Coil14HitCurrent_GET : MESSAGE;
        MessageParameters(ServiceCode := 16#000e, DestinationTag := STA_Coil14HitCurrent_GET_VAL, ...)
   STA_Coil14HitCurrent_GET_VAL : INT;
   STA_Coil14HitCurrent_TRG_GET : BOOL;
   STA_Coil14HitPower_GET : MESSAGE;
        MessageParameters(ServiceCode := 16#000e, DestinationTag := STA_Coil14HitPower_GET_VAL, ...)
   STA_Coil14HitPower_GET_VAL : INT;
   STA_Coil14HitPower_TRG_GET : BOOL;
   STA_Coil14HoldCurrent_GET : MESSAGE;
        MessageParameters(ServiceCode := 16#000e, DestinationTag := STA_Coil14HoldCurrent_GET_VAL, ...)
   STA_Coil14HoldCurrent_GET_VAL : INT;
   STA_Coil14HoldCurrent_TRG_GET : BOOL;
   STA_Coil14HoldPower_GET : MESSAGE;
        MessageParameters(ServiceCode := 16#000e, DestinationTag := STA_Coil14HoldPower_Get_VAL, ...)
   STA_Coil14HoldPower_Get_VAL : INT;
   STA_Coil14HoldPower_SET : MESSAGE;
        MessageParameters(ServiceCode := 16#0010, LocalElement := STA_Coil14HoldPower_Set_VAL, ...)
   STA_Coil14HoldPower_Set_VAL : INT;
   STA_Coil14HoldPower_TRG_GET : BOOL;
   STA_Coil14HoldPower_TRG_SET : BOOL;
   STA_Coil14HoldVolage_GET : MESSAGE;
        MessageParameters(ServiceCode := 16#000e, DestinationTag := STA_Coil14HoldVolage_Get_VAL, ...)
   STA_Coil14HoldVolage_Get_VAL : INT;
   STA_Coil14HoldVolage_SET : MESSAGE;
        MessageParameters(ServiceCode := 16#0010, LocalElement := STA_Coil14HoldVolage_Set_VAL, ...)
   STA_Coil14HoldVolage_Set_VAL : INT;
   STA_Coil14HoldVolage_TRG_GET : BOOL;
   STA_Coil14HoldVolage_TRG_SET : BOOL;
   STA_DV_ERROR_STATUS_GET : MESSAGE;
        MessageParameters(ServiceCode := 16#000e, DestinationTag := STA_DV_ERROR_STATUS_GET_VAL, ...)
   STA_DV_ERROR_STATUS_GET_VAL : UINT;
   STA_DV_ERROR_STATUS_TRG_GET : BOOL;
   STA_ExhaustPresHysteresis_GET : MESSAGE;
        MessageParameters(ServiceCode := 16#000e, DestinationTag := STA_ExhaustPresHysteresis_Get_VAL, ...)
   STA_ExhaustPresHysteresis_Get_VAL : INT;
   STA_ExhaustPresHysteresis_SET : MESSAGE;
        MessageParameters(ServiceCode := 16#0010, LocalElement := STA_ExhaustPresHysteresis_Set_VAL, ...)
   STA_ExhaustPresHysteresis_Set_VAL : INT;
   STA_ExhaustPresHysteresis_TRG_GET : BOOL;
   STA_ExhaustPresHysteresis_TRG_SET : BOOL;
   STA_FAULTEVNTBITS_GET : MESSAGE;
        MessageParameters(ServiceCode := 16#000e, DestinationTag := STA_FAULTEVNTBITS_GET_VAL, ...)
   STA_FAULTEVNTBITS_GET_VAL : UDINT;
   STA_FAULTEVNTBITS_TRG_GET : BOOL;
   STA_FAULTEVNTCOUNT_GET : MESSAGE;
        MessageParameters(ServiceCode := 16#000e, DestinationTag := STA_FAULTEVNTCOUNT_GET_VAL, ...)
   STA_FAULTEVNTCOUNT_GET_VAL : UINT;
   STA_FAULTEVNTCOUNT_TRG_GET : BOOL;
   STA_IDENT_DEVICETYPE_GET : MESSAGE;
        MessageParameters(ServiceCode := 16#000e, DestinationTag := STA_IDENT_DEVICETYPE_GET_VAL, ...)
   STA_IDENT_DEVICETYPE_GET_VAL : UDINT;
   STA_IDENT_DEVICETYPE_TRG_GET : BOOL;
   STA_INTR_IDENT_DEVICEID_GET : MESSAGE;
        MessageParameters(ServiceCode := 16#000e, DestinationTag := STA_INTR_IDENT_DEVICEID_GET_VAL, ...)
   STA_INTR_IDENT_DEVICEID_GET_VAL : UDINT;
   STA_INTR_IDENT_DEVICEID_TRG_GET : BOOL;
   STA_INTR_IDENT_DEVICENAME_GET : MESSAGE;
        MessageParameters(ServiceCode := 16#000e, DestinationTag := STA_INTR_IDENT_DEVICENAME_GET_VAL, ...)
   STA_INTR_IDENT_DEVICENAME_GET_VAL : STR_20;
   STA_INTR_IDENT_DEVICENAME_TRG_GET : BOOL;
   STA_INTR_IDENT_HWREV_GET : MESSAGE;
        MessageParameters(ServiceCode := 16#000e, DestinationTag := STA_INTR_IDENT_HWREV_GET_VAL, ...)
   STA_INTR_IDENT_HWREV_GET_VAL : STR_20;
   STA_INTR_IDENT_HWREV_TRG_GET : BOOL;
   STA_INTR_IDENT_SERIALNO_GET : MESSAGE;
        MessageParameters(ServiceCode := 16#000e, DestinationTag := STA_INTR_IDENT_SERIALNO_GET_VAL, ...)
   STA_INTR_IDENT_SERIALNO_GET_VAL : STR_20;
   STA_INTR_IDENT_SERIALNO_TRG_GET : BOOL;
   STA_INTR_IDENT_SWPARTNO_GET : MESSAGE;
        MessageParameters(ServiceCode := 16#000e, DestinationTag := STA_INTR_IDENT_SWPARTNO_GET_VAL, ...)
   STA_INTR_IDENT_SWPARTNO_GET_VAL : STR_20;
   STA_INTR_IDENT_SWPARTNO_TRG_GET : BOOL;
   STA_INTR_IDENT_SWREV_GET : MESSAGE;
        MessageParameters(ServiceCode := 16#000e, DestinationTag := STA_INTR_IDENT_SWREV_GET_VAL, ...)
   STA_INTR_IDENT_SWREV_GET_VAL : STR_20;
   STA_INTR_IDENT_SWREV_TRG_GET : BOOL;
   STA_INTR_IDENT_VARIANTID_GET : MESSAGE;
        MessageParameters(ServiceCode := 16#000e, DestinationTag := STA_INTR_IDENT_VARIANTID_GET_VAL, ...)
   STA_INTR_IDENT_VARIANTID_GET_VAL : STR_20;
   STA_INTR_IDENT_VARIANTID_TRG_GET : BOOL;
   STA_INTR_IDENT_VENDORID_GET : MESSAGE;
        MessageParameters(ServiceCode := 16#000e, DestinationTag := STA_INTR_IDENT_VENDORID_GET_VAL, ...)
   STA_INTR_IDENT_VENDORID_GET_VAL : UDINT;
   STA_INTR_IDENT_VENDORID_TRG_GET : BOOL;
   STA_INTR_IDENT_VENDORNAME_GET : MESSAGE;
        MessageParameters(ServiceCode := 16#000e, DestinationTag := STA_INTR_IDENT_VENDORNAME_GET_VAL, ...)
   STA_INTR_IDENT_VENDORNAME_GET_VAL : STR_20;
   STA_INTR_IDENT_VENDORNAME_TRG_GET : BOOL;
   STA_MaxApplPressure_GET : MESSAGE;
        MessageParameters(ServiceCode := 16#000e, DestinationTag := STA_MaxApplPressure_Get_VAL, ...)
   STA_MaxApplPressure_Get_VAL : INT;
   STA_MaxApplPressure_SET : MESSAGE;
        MessageParameters(ServiceCode := 16#0010, LocalElement := STA_MaxApplPressure_Set_VAL, ...)
   STA_MaxApplPressure_Set_VAL : INT;
   STA_MaxApplPressure_TRG_GET : BOOL;
   STA_MaxApplPressure_TRG_SET : BOOL;
   STA_MeasuredAuxVolt_GET : MESSAGE;
        MessageParameters(ServiceCode := 16#000e, DestinationTag := STA_MeasuredAuxVolt_GET_VAL, ...)
   STA_MeasuredAuxVolt_GET_VAL : INT;
   STA_MeasuredAuxVolt_TRG_GET : BOOL;
   STA_MinApplPressure_GET : MESSAGE;
        MessageParameters(ServiceCode := 16#000e, DestinationTag := STA_MinApplPressure_Get_VAL, ...)
   STA_MinApplPressure_Get_VAL : INT;
   STA_MinApplPressure_SET : MESSAGE;
        MessageParameters(ServiceCode := 16#0010, LocalElement := STA_MinApplPressure_Set_VAL, ...)
   STA_MinApplPressure_Set_VAL : INT;
   STA_MinApplPressure_TRG_GET : BOOL;
   STA_MinApplPressure_TRG_SET : BOOL;
   STA_OPERATIONTIME_HR_GET : MESSAGE;
        MessageParameters(ServiceCode := 16#000e, DestinationTag := STA_OPERATIONTIME_HR_GET_VAL, ...)
   STA_OPERATIONTIME_HR_GET_VAL : UDINT;
   STA_OPERATIONTIME_HR_TRG_GET : BOOL;
   STA_OPERATIONTIME_MIN_GET : MESSAGE;
        MessageParameters(ServiceCode := 16#000e, DestinationTag := STA_OPERATIONTIME_MIN_GET_VAL, ...)
   STA_OPERATIONTIME_MIN_GET_VAL : UINT;
   STA_OPERATIONTIME_MIN_TRG_GET : BOOL;
   STA_Port2ApplPressCyclRating_GET : MESSAGE;
        MessageParameters(ServiceCode := 16#000e, DestinationTag := STA_Port2ApplPressCyclRating_Get_VAL, ...)
   STA_Port2ApplPressCyclRating_Get_VAL : UDINT;
   STA_Port2ApplPressCyclRating_SET : MESSAGE;
        MessageParameters(ServiceCode := 16#0010, LocalElement := STA_Port2ApplPressCyclRating_Set_VAL, ...)
   STA_Port2ApplPressCyclRating_Set_VAL : UDINT;
   STA_Port2ApplPressCyclRating_TRG_GET : BOOL;
   STA_Port2ApplPressCyclRating_TRG_SET : BOOL;
   STA_Port2MesrdPressure_GET : MESSAGE;
        MessageParameters(ServiceCode := 16#000e, DestinationTag := STA_Port2MesrdPressure_GET_VAL, ...)
   STA_Port2MesrdPressure_GET_VAL : INT;
   STA_Port2MesrdPressure_TRG_GET : BOOL;
   STA_Port2PressCycleCounter_GET : MESSAGE;
        MessageParameters(ServiceCode := 16#000e, DestinationTag := STA_Port2PressCycleCounter_GET_VAL, ...)
   STA_Port2PressCycleCounter_GET_VAL : UDINT;
   STA_Port2PressCycleCounter_TRG_GET : BOOL;
   STA_Port2PressMonitorDly_GET : MESSAGE;
        MessageParameters(ServiceCode := 16#000e, DestinationTag := STA_Port2PressMonitorDly_Get_VAL, ...)
   STA_Port2PressMonitorDly_Get_VAL : UINT;
   STA_Port2PressMonitorDly_SET : MESSAGE;
        MessageParameters(ServiceCode := 16#0010, LocalElement := STA_Port2PressMonitorDly_Set_VAL, ...)
   STA_Port2PressMonitorDly_Set_VAL : UINT;
   STA_Port2PressMonitorDly_TRG_GET : BOOL;
   STA_Port2PressMonitorDly_TRG_SET : BOOL;
   STA_Port4ApplPressCyclRating_GET : MESSAGE;
        MessageParameters(ServiceCode := 16#000e, DestinationTag := STA_Port4ApplPressCyclRating_Get_VAL, ...)
   STA_Port4ApplPressCyclRating_Get_VAL : UDINT;
   STA_Port4ApplPressCyclRating_SET : MESSAGE;
        MessageParameters(ServiceCode := 16#0010, LocalElement := STA_Port4ApplPressCyclRating_Set_VAL, ...)
   STA_Port4ApplPressCyclRating_Set_VAL : UDINT;
   STA_Port4ApplPressCyclRating_TRG_GET : BOOL;
   STA_Port4ApplPressCyclRating_TRG_SET : BOOL;
   STA_Port4MesrdPressure_GET : MESSAGE;
        MessageParameters(ServiceCode := 16#000e, DestinationTag := STA_Port4MesrdPressure_GET_VAL, ...)
   STA_Port4MesrdPressure_GET_VAL : INT;
   STA_Port4MesrdPressure_TRG_GET : BOOL;
   STA_Port4PressCycleCounter_GET : MESSAGE;
        MessageParameters(ServiceCode := 16#000e, DestinationTag := STA_Port4PressCycleCounter_GET_VAL, ...)
   STA_Port4PressCycleCounter_GET_VAL : UDINT;
   STA_Port4PressCycleCounter_TRG_GET : BOOL;
   STA_Port4PressMonitorDly_GET : MESSAGE;
        MessageParameters(ServiceCode := 16#000e, DestinationTag := STA_Port4PressMonitorDly_Get_VAL, ...)
   STA_Port4PressMonitorDly_Get_VAL : UINT;
   STA_Port4PressMonitorDly_SET : MESSAGE;
        MessageParameters(ServiceCode := 16#0010, LocalElement := STA_Port4PressMonitorDly_set_VAL, ...)
   STA_Port4PressMonitorDly_set_VAL : UINT;
   STA_Port4PressMonitorDly_TRG_GET : BOOL;
   STA_Port4PressMonitorDly_TRG_SET : BOOL;
   STA_PWRONTIME_HR_GET : MESSAGE;
        MessageParameters(ServiceCode := 16#000e, DestinationTag := STA_PWRONTIME_HR_GET_VAL, ...)
   STA_PWRONTIME_HR_GET_VAL : UDINT;
   STA_PWRONTIME_HR_TRG_GET : BOOL;
   STA_PWRONTIME_MIN_GET : MESSAGE;
        MessageParameters(ServiceCode := 16#000e, DestinationTag := STA_PWRONTIME_MIN_GET_VAL, ...)
   STA_PWRONTIME_MIN_GET_VAL : UINT;
   STA_PWRONTIME_MIN_TRG_GET : BOOL;
   STA_RatedAuxVoltHyst_GET : MESSAGE;
        MessageParameters(ServiceCode := 16#000e, DestinationTag := STA_RatedAuxVoltHyst_Get_VAL, ...)
   STA_RatedAuxVoltHyst_Get_VAL : INT;
   STA_RatedAuxVoltHyst_SET : MESSAGE;
        MessageParameters(ServiceCode := 16#0010, LocalElement := STA_RatedAuxVoltHyst_Set_VAL, ...)
   STA_RatedAuxVoltHyst_Set_VAL : INT;
   STA_RatedAuxVoltHyst_TRG_GET : BOOL;
   STA_RatedAuxVoltHyst_TRG_SET : BOOL;
   STA_Valve12ApplCyclRating_GET : MESSAGE;
        MessageParameters(ServiceCode := 16#000e, DestinationTag := STA_Valve12ApplCyclRating_Get_VAL, ...)
   STA_Valve12ApplCyclRating_Get_VAL : UDINT;
   STA_Valve12ApplCyclRating_SET : MESSAGE;
        MessageParameters(ServiceCode := 16#0010, LocalElement := STA_Valve12ApplCyclRating_Set_VAL, ...)
   STA_Valve12ApplCyclRating_Set_VAL : UDINT;
   STA_Valve12ApplCyclRating_TRG_GET : BOOL;
   STA_Valve12ApplCyclRating_TRG_SET : BOOL;
   STA_Valve12CycleCounter_GET : MESSAGE;
        MessageParameters(ServiceCode := 16#000e, DestinationTag := STA_Valve12CycleCounter_GET_VAL, ...)
   STA_Valve12CycleCounter_GET_VAL : UDINT;
   STA_Valve12CycleCounter_TRG_GET : BOOL;
   STA_Valve14ApplCyclRating_GET : MESSAGE;
        MessageParameters(ServiceCode := 16#000e, DestinationTag := STA_Valve14ApplCyclRating_Get_VAL, ...)
   STA_Valve14ApplCyclRating_Get_VAL : UDINT;
   STA_Valve14ApplCyclRating_SET : MESSAGE;
        MessageParameters(ServiceCode := 16#0010, LocalElement := STA_Valve14ApplCyclRating_Set_VAL, ...)
   STA_Valve14ApplCyclRating_Set_VAL : UDINT;
   STA_Valve14ApplCyclRating_TRG_GET : BOOL;
   STA_Valve14ApplCyclRating_TRG_SET : BOOL;
   STA_Valve14CycleCounter_GET : MESSAGE;
        MessageParameters(ServiceCode := 16#000e, DestinationTag := STA_Valve14CycleCounter_GET_VAL, ...)
   STA_Valve14CycleCounter_GET_VAL : UDINT;
   STA_Valve14CycleCounter_TRG_GET : BOOL;
   STA_ValveSlice12Side_GET : MESSAGE;
        MessageParameters(ServiceCode := 16#000e, DestinationTag := STA_ValveSlice12Side_Get_VAL, ...)
   STA_ValveSlice12Side_Get_VAL : UINT;
   STA_ValveSlice12Side_SET : MESSAGE;
        MessageParameters(ServiceCode := 16#0010, LocalElement := STA_ValveSlice12Side_Set_VAL, ...)
   STA_ValveSlice12Side_Set_VAL : UINT;
   STA_ValveSlice12Side_TRG_GET : BOOL;
   STA_ValveSlice12Side_TRG_SET : BOOL;
   STA_ValveSliceFunction_GET : MESSAGE;
        MessageParameters(ServiceCode := 16#000e, DestinationTag := STA_ValveSliceFunction_Get_VAL, ...)
   STA_ValveSliceFunction_Get_VAL : UINT;
   STA_ValveSliceFunction_SET : MESSAGE;
        MessageParameters(ServiceCode := 16#0010, LocalElement := STA_ValveSliceFunction_Set_VAL, ...)
   STA_ValveSliceFunction_Set_VAL : UINT;
   STA_ValveSliceFunction_TRG_GET : BOOL;
   STA_ValveSliceFunction_TRG_SET : BOOL;
   STA_WARNEVNTBITS_GET : MESSAGE;
        MessageParameters(ServiceCode := 16#000e, DestinationTag := STA_WARNEVNTBITS_GET_VAL, ...)
   STA_WARNEVNTBITS_GET_VAL : UDINT;
   STA_WARNEVNTBITS_TRG_GET : BOOL;
   STA_WARNEVNTCOUNT_GET : MESSAGE;
        MessageParameters(ServiceCode := 16#000e, DestinationTag := STA_WARNEVNTCOUNT_GET_VAL, ...)
   STA_WARNEVNTCOUNT_GET_VAL : UINT;
   STA_WARNEVNTCOUNT_TRG_GET : BOOL;
   STA_WARNSTSBITS_GET : MESSAGE;
        MessageParameters(ServiceCode := 16#000e, DestinationTag := STA_WARNSTSBITS_GET_VAL, ...)
   STA_WARNSTSBITS_GET_VAL : UDINT;
   STA_WARNSTSBITS_TRG_GET : BOOL;
   up_counter : COUNTER;
   VA_VOLTAGE_GET : MESSAGE;
        MessageParameters(ServiceCode := 16#000e, DestinationTag := VA_VOLTAGE_GET_VAL, ...)
   VA_VOLTAGE_GET_VAL : UDINT;
   VA_VOLTAGE_TRG_GET : BOOL;
   valve_on : BOOL;
   VB_VOLTAGE_GET : MESSAGE;
        MessageParameters(ServiceCode := 16#000e, DestinationTag := VB_VOLTAGE_GET_VAL, ...)
   VB_VOLTAGE_GET_VAL : UDINT;
   VB_VOLTAGE_TRG_GET : BOOL;
END_VAR
VAR {public}
   Diag_Valve_Err_Status : ALIAS FOR VRQx:I.Diag_Valve_Err_Status;
   Digital_Input_ch1 : ALIAS FOR VRQx:I.Ditigal_Input_Ch1_to_Ch4_0.0;
   Digital_Input_ch2 : ALIAS FOR VRQx:I.Ditigal_Input_Ch1_to_Ch4_0.1;
   Digital_Input_ch3 : ALIAS FOR VRQx:I.Ditigal_Input_Ch1_to_Ch4_0.2;
   Digital_Input_ch4 : ALIAS FOR VRQx:I.Ditigal_Input_Ch1_to_Ch4_0.3;
   Digital_Output_ch1 : ALIAS FOR VRQx:O.Data[0].0;
   Digital_Output_ch2 : ALIAS FOR VRQx:O.Data[0].1;
   Digital_Output_ch3 : ALIAS FOR VRQx:O.Data[0].2;
   Digital_Output_ch4 : ALIAS FOR VRQx:O.Data[0].3;
   DIO_Module_Input_Error : ALIAS FOR VRQx:I.DIO_Module_ErrorStatus_0.0;
   DIO_Module_Output_Error : ALIAS FOR VRQx:I.DIO_Module_ErrorStatus_0.1;
   DIO_Module_Self_test_error : ALIAS FOR VRQx:I.DIO_Module_ErrorStatus_0.4;
   DIO_Module_VA_Over_Voltage_Under_Volta : ALIAS FOR VRQx:I.DIO_Module_ErrorStatus_0.2;
   DIO_Module_VB_Over_Voltage_Under_Volta : ALIAS FOR VRQx:I.DIO_Module_ErrorStatus_0.3;
   ISEM_DV_PDI_ch1 : ALIAS FOR VRQx:I.ISEM_DV_PDI_ch1;
   ISEM_DV_PDI_ch2 : ALIAS FOR VRQx:I.ISEM_DV_PDI_ch2;
   ISEM_DV_PDI_ch3 : ALIAS FOR VRQx:I.ISEM_DV_PDI_ch3;
   ISEM_DV_PDI_ch4 : ALIAS FOR VRQx:I.ISEM_DV_PDI_ch4;
   ISEM_DV_PDI_ch5 : ALIAS FOR VRQx:I.ISEM_DV_PDI_ch5;
   ISEM_DV_PDI_ch6 : ALIAS FOR VRQx:I.ISEM_DV_PDI_ch6;
   ISEM_DV_PDI_ch7 : ALIAS FOR VRQx:I.ISEM_DV_PDI_ch7;
   ISEM_DV_PDI_ch8 : ALIAS FOR VRQx:I.ISEM_DV_PDI_ch8;
   ISEM_PDI : ALIAS FOR VRQx:I.ISEM_PDI;
   Output_Port_Pressure : ALIAS FOR VRQx:I.Output_Port_Pressure;
   PROP_PDI : ALIAS FOR VRQx:I.PROP_PDI;
   PROP_PDO_Higher_Byte : ALIAS FOR VRQx:O.Data[4];
   PROP_PDO_Lower_Byte : ALIAS FOR VRQx:O.Data[3];
   Prop_Set_Point_Pressure_Higher_Byte : ALIAS FOR VRQx:O.Data[6];
   Prop_Set_Point_Pressure_Lower_Byte : ALIAS FOR VRQx:O.Data[5];
   Station_1A : ALIAS FOR VRQx:O.Data[1].7;
   Station_1B : ALIAS FOR VRQx:O.Data[1].6;
   Station_2A : ALIAS FOR VRQx:O.Data[1].5;
   Station_2B : ALIAS FOR VRQx:O.Data[1].4;
   Station_3A : ALIAS FOR VRQx:O.Data[1].3;
   Station_3B : ALIAS FOR VRQx:O.Data[1].2;
   Station_4A : ALIAS FOR VRQx:O.Data[1].1;
   Station_4B : ALIAS FOR VRQx:O.Data[1].0;
   Station_5A : ALIAS FOR VRQx:O.Data[2].7;
   Station_5B : ALIAS FOR VRQx:O.Data[2].6;
   Station_6A : ALIAS FOR VRQx:O.Data[2].5;
   Station_6B : ALIAS FOR VRQx:O.Data[2].4;
   Station_7A : ALIAS FOR VRQx:O.Data[2].3;
   Station_7B : ALIAS FOR VRQx:O.Data[2].2;
   Station_8A : ALIAS FOR VRQx:O.Data[2].1;
   Station_8B : ALIAS FOR VRQx:O.Data[2].0;
   TLE_Diagnostics_Error_Status : ALIAS FOR VRQx:I.TLE_Diagnostics_Err_Status;
END_VAR

ROUTINE MainRoutine   (* ladder *)
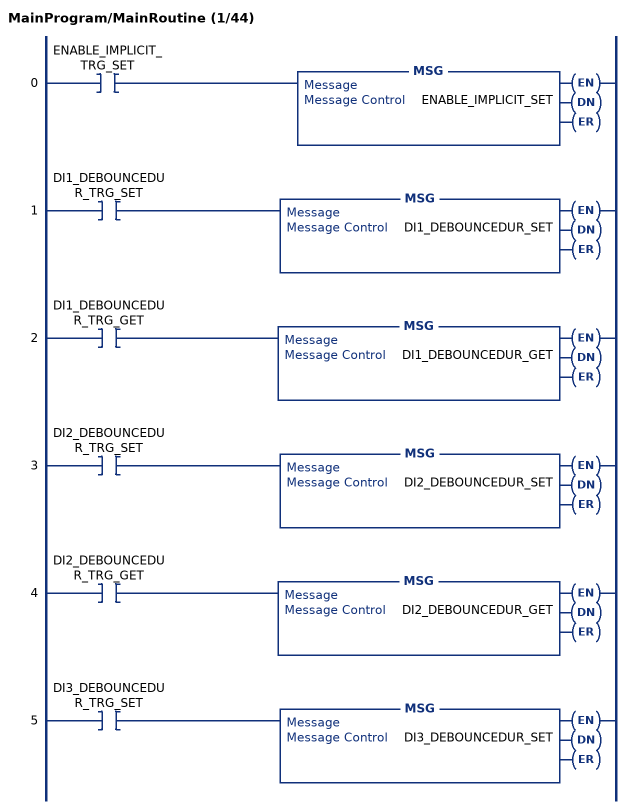
   0: XIC(ENABLE_IMPLICIT_TRG_SET)MSG(ENABLE_IMPLICIT_SET);
   1: XIC(DI1_DEBOUNCEDUR_TRG_SET)MSG(DI1_DEBOUNCEDUR_SET);
   2: XIC(DI1_DEBOUNCEDUR_TRG_GET)MSG(DI1_DEBOUNCEDUR_GET);
   3: XIC(DI2_DEBOUNCEDUR_TRG_SET)MSG(DI2_DEBOUNCEDUR_SET);
   4: XIC(DI2_DEBOUNCEDUR_TRG_GET)MSG(DI2_DEBOUNCEDUR_GET);
   5: XIC(DI3_DEBOUNCEDUR_TRG_SET)MSG(DI3_DEBOUNCEDUR_SET);
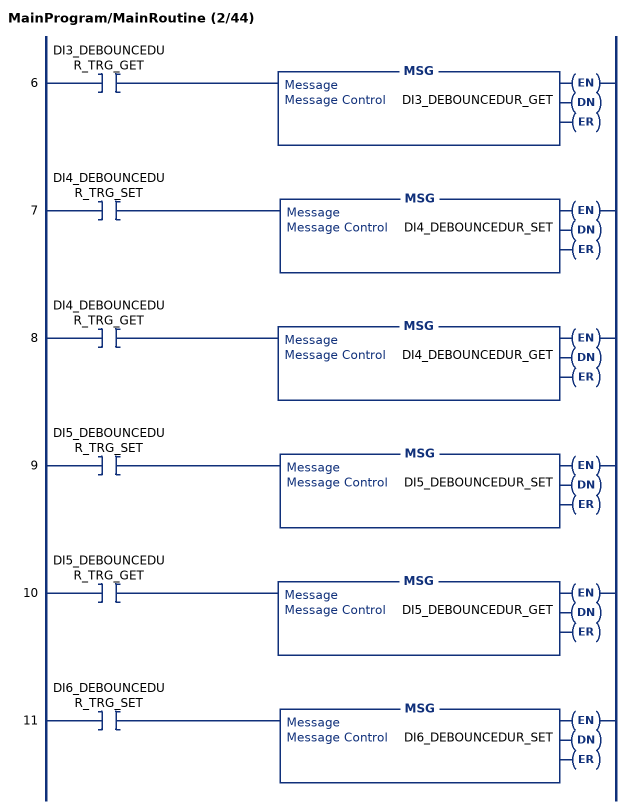
   6: XIC(DI3_DEBOUNCEDUR_TRG_GET)MSG(DI3_DEBOUNCEDUR_GET);
   7: XIC(DI4_DEBOUNCEDUR_TRG_SET)MSG(DI4_DEBOUNCEDUR_SET);
   8: XIC(DI4_DEBOUNCEDUR_TRG_GET)MSG(DI4_DEBOUNCEDUR_GET);
   9: XIC(DI5_DEBOUNCEDUR_TRG_SET)MSG(DI5_DEBOUNCEDUR_SET);
   10: XIC(DI5_DEBOUNCEDUR_TRG_GET)MSG(DI5_DEBOUNCEDUR_GET);
   11: XIC(DI6_DEBOUNCEDUR_TRG_SET)MSG(DI6_DEBOUNCEDUR_SET);
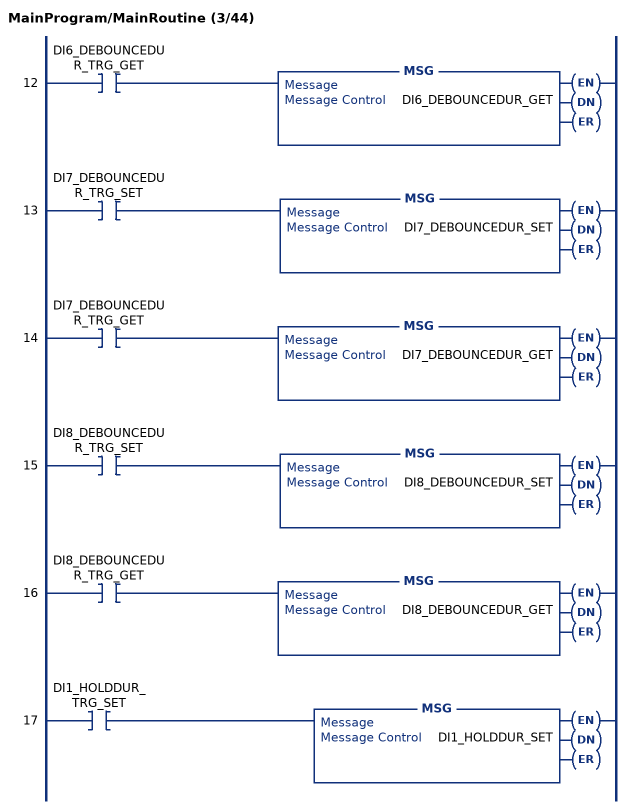
   12: XIC(DI6_DEBOUNCEDUR_TRG_GET)MSG(DI6_DEBOUNCEDUR_GET);
   13: XIC(DI7_DEBOUNCEDUR_TRG_SET)MSG(DI7_DEBOUNCEDUR_SET);
   14: XIC(DI7_DEBOUNCEDUR_TRG_GET)MSG(DI7_DEBOUNCEDUR_GET);
   15: XIC(DI8_DEBOUNCEDUR_TRG_SET)MSG(DI8_DEBOUNCEDUR_SET);
   16: XIC(DI8_DEBOUNCEDUR_TRG_GET)MSG(DI8_DEBOUNCEDUR_GET);
   17: XIC(DI1_HOLDDUR_TRG_SET)MSG(DI1_HOLDDUR_SET);
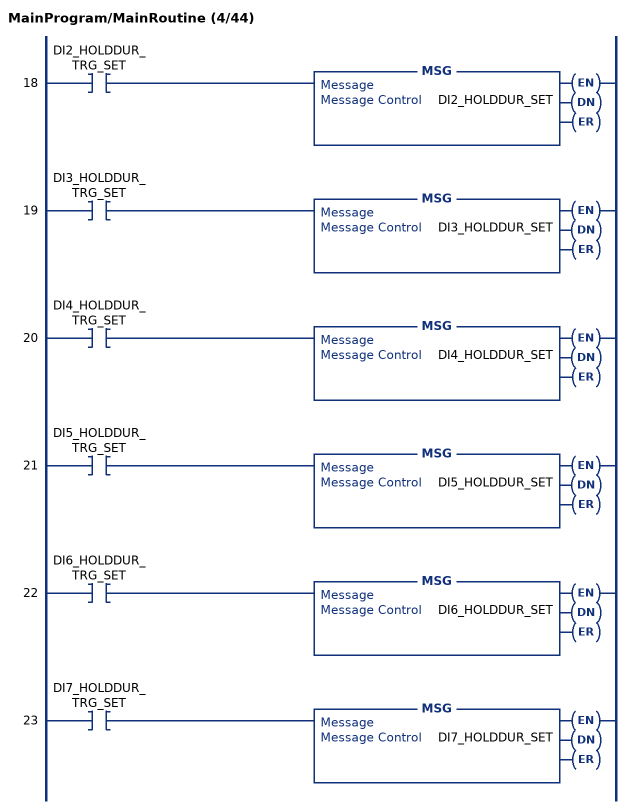
   18: XIC(DI2_HOLDDUR_TRG_SET)MSG(DI2_HOLDDUR_SET);
   19: XIC(DI3_HOLDDUR_TRG_SET)MSG(DI3_HOLDDUR_SET);
   20: XIC(DI4_HOLDDUR_TRG_SET)MSG(DI4_HOLDDUR_SET);
   21: XIC(DI5_HOLDDUR_TRG_SET)MSG(DI5_HOLDDUR_SET);
   22: XIC(DI6_HOLDDUR_TRG_SET)MSG(DI6_HOLDDUR_SET);
   23: XIC(DI7_HOLDDUR_TRG_SET)MSG(DI7_HOLDDUR_SET);
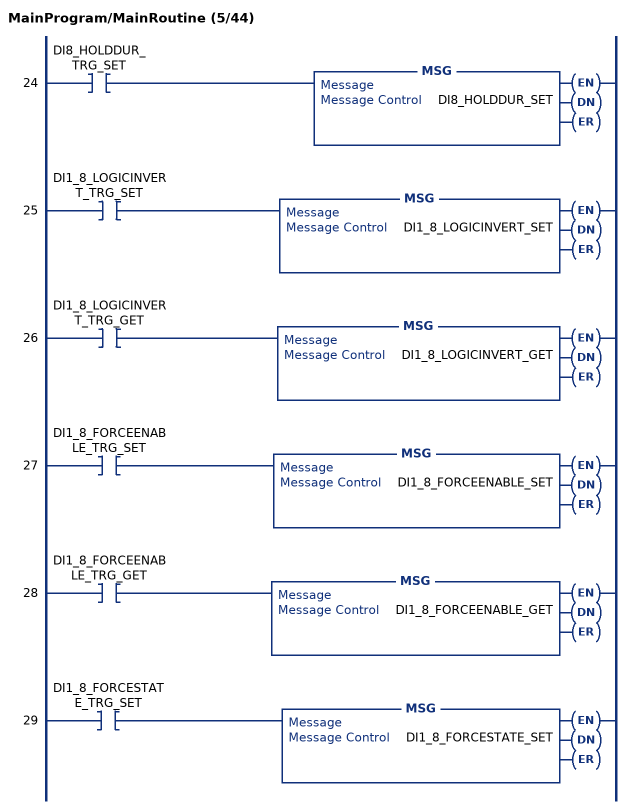
   24: XIC(DI8_HOLDDUR_TRG_SET)MSG(DI8_HOLDDUR_SET);
   25: XIC(DI1_8_LOGICINVERT_TRG_SET)MSG(DI1_8_LOGICINVERT_SET);
   26: XIC(DI1_8_LOGICINVERT_TRG_GET)MSG(DI1_8_LOGICINVERT_GET);
   27: XIC(DI1_8_FORCEENABLE_TRG_SET)MSG(DI1_8_FORCEENABLE_SET);
   28: XIC(DI1_8_FORCEENABLE_TRG_GET)MSG(DI1_8_FORCEENABLE_GET);
   29: XIC(DI1_8_FORCESTATE_TRG_SET)MSG(DI1_8_FORCESTATE_SET);
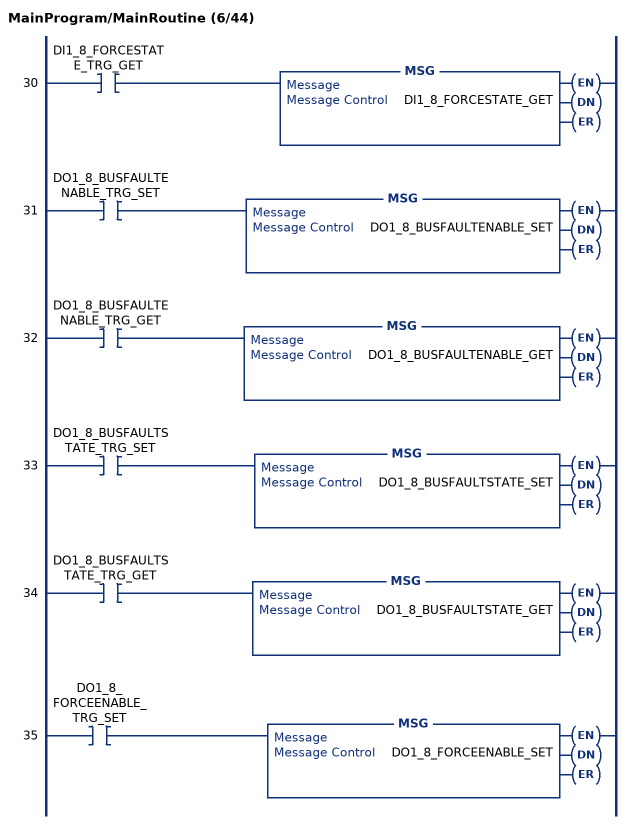
   30: XIC(DI1_8_FORCESTATE_TRG_GET)MSG(DI1_8_FORCESTATE_GET);
   31: XIC(DO1_8_BUSFAULTENABLE_TRG_SET)MSG(DO1_8_BUSFAULTENABLE_SET);
   32: XIC(DO1_8_BUSFAULTENABLE_TRG_GET)MSG(DO1_8_BUSFAULTENABLE_GET);
   33: XIC(DO1_8_BUSFAULTSTATE_TRG_SET)MSG(DO1_8_BUSFAULTSTATE_SET);
   34: XIC(DO1_8_BUSFAULTSTATE_TRG_GET)MSG(DO1_8_BUSFAULTSTATE_GET);
   35: XIC(DO1_8_FORCEENABLE_TRG_SET)MSG(DO1_8_FORCEENABLE_SET);
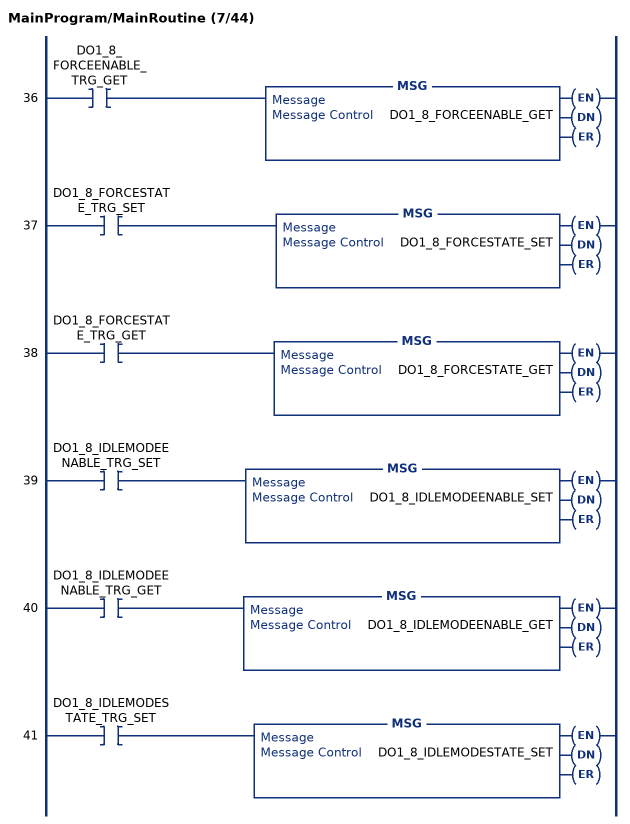
   36: XIC(DO1_8_FORCEENABLE_TRG_GET)MSG(DO1_8_FORCEENABLE_GET);
   37: XIC(DO1_8_FORCESTATE_TRG_SET)MSG(DO1_8_FORCESTATE_SET);
   38: XIC(DO1_8_FORCESTATE_TRG_GET)MSG(DO1_8_FORCESTATE_GET);
   39: XIC(DO1_8_IDLEMODEENABLE_TRG_SET)MSG(DO1_8_IDLEMODEENABLE_SET);
   40: XIC(DO1_8_IDLEMODEENABLE_TRG_GET)MSG(DO1_8_IDLEMODEENABLE_GET);
   41: XIC(DO1_8_IDLEMODESTATE_TRG_SET)MSG(DO1_8_IDLEMODESTATE_SET);
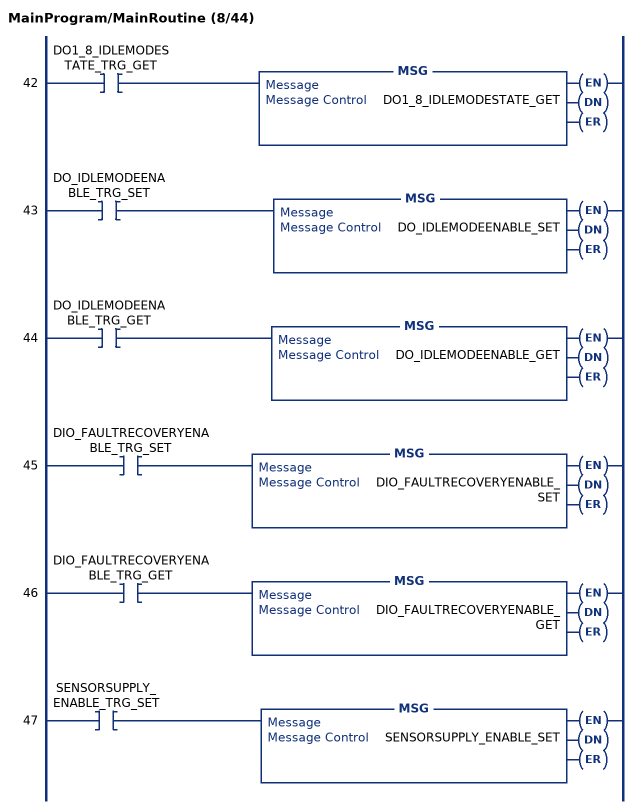
   42: XIC(DO1_8_IDLEMODESTATE_TRG_GET)MSG(DO1_8_IDLEMODESTATE_GET);
   43: XIC(DO_IDLEMODEENABLE_TRG_SET)MSG(DO_IDLEMODEENABLE_SET);
   44: XIC(DO_IDLEMODEENABLE_TRG_GET)MSG(DO_IDLEMODEENABLE_GET);
   45: XIC(DIO_FAULTRECOVERYENABLE_TRG_SET)MSG(DIO_FAULTRECOVERYENABLE_SET);
   46: XIC(DIO_FAULTRECOVERYENABLE_TRG_GET)MSG(DIO_FAULTRECOVERYENABLE_GET);
   47: XIC(SENSORSUPPLY_ENABLE_TRG_SET)MSG(SENSORSUPPLY_ENABLE_SET);
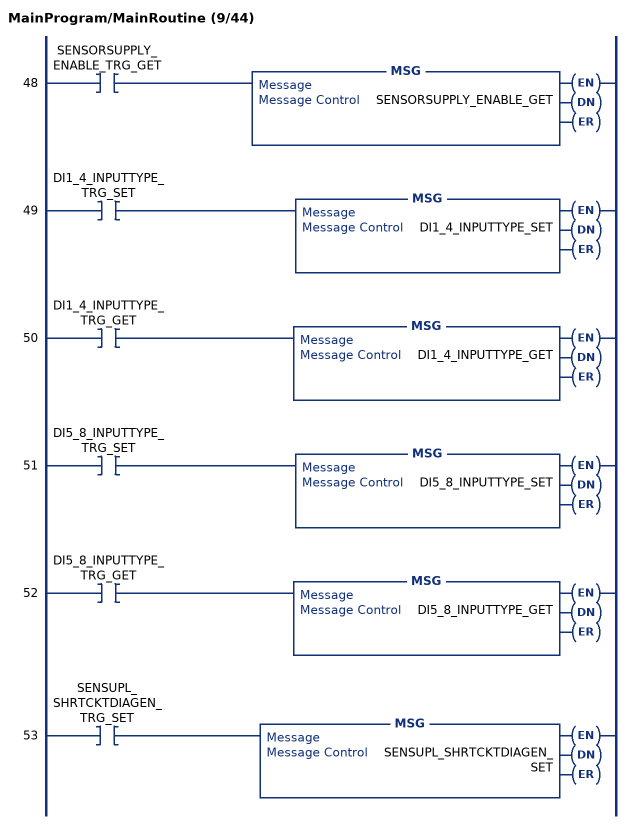
   48: XIC(SENSORSUPPLY_ENABLE_TRG_GET)MSG(SENSORSUPPLY_ENABLE_GET);
   49: XIC(DI1_4_INPUTTYPE_TRG_SET)MSG(DI1_4_INPUTTYPE_SET);
   50: XIC(DI1_4_INPUTTYPE_TRG_GET)MSG(DI1_4_INPUTTYPE_GET);
   51: XIC(DI5_8_INPUTTYPE_TRG_SET)MSG(DI5_8_INPUTTYPE_SET);
   52: XIC(DI5_8_INPUTTYPE_TRG_GET)MSG(DI5_8_INPUTTYPE_GET);
   53: XIC(SENSUPL_SHRTCKTDIAGEN_TRG_SET)MSG(SENSUPL_SHRTCKTDIAGEN_SET);
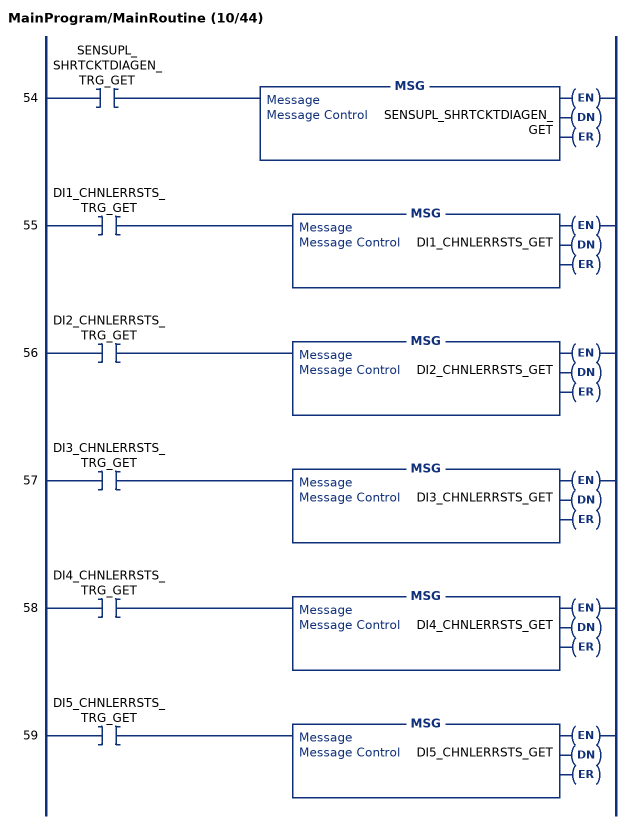
   54: XIC(SENSUPL_SHRTCKTDIAGEN_TRG_GET)MSG(SENSUPL_SHRTCKTDIAGEN_GET);
   55: XIC(DI1_CHNLERRSTS_TRG_GET)MSG(DI1_CHNLERRSTS_GET);
   56: XIC(DI2_CHNLERRSTS_TRG_GET)MSG(DI2_CHNLERRSTS_GET);
   57: XIC(DI3_CHNLERRSTS_TRG_GET)MSG(DI3_CHNLERRSTS_GET);
   58: XIC(DI4_CHNLERRSTS_TRG_GET)MSG(DI4_CHNLERRSTS_GET);
   59: XIC(DI5_CHNLERRSTS_TRG_GET)MSG(DI5_CHNLERRSTS_GET);
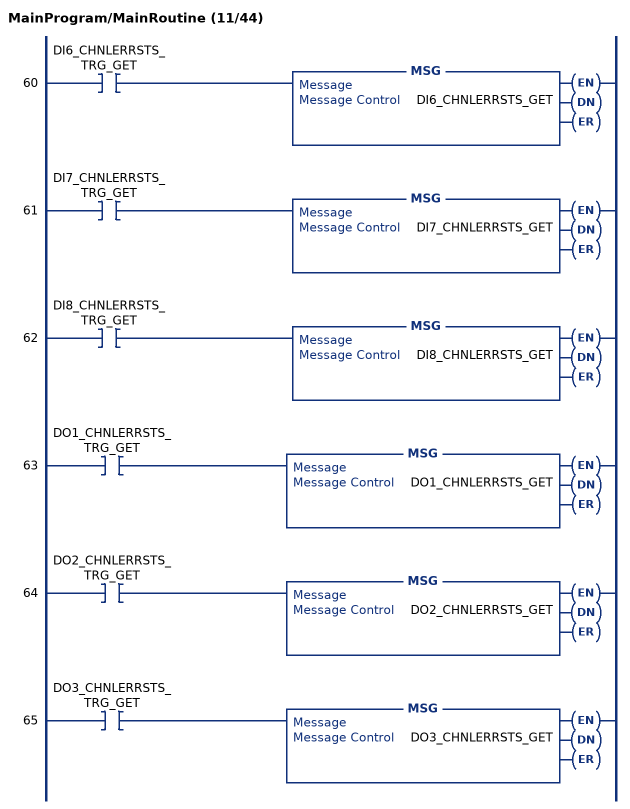
   60: XIC(DI6_CHNLERRSTS_TRG_GET)MSG(DI6_CHNLERRSTS_GET);
   61: XIC(DI7_CHNLERRSTS_TRG_GET)MSG(DI7_CHNLERRSTS_GET);
   62: XIC(DI8_CHNLERRSTS_TRG_GET)MSG(DI8_CHNLERRSTS_GET);
   63: XIC(DO1_CHNLERRSTS_TRG_GET)MSG(DO1_CHNLERRSTS_GET);
   64: XIC(DO2_CHNLERRSTS_TRG_GET)MSG(DO2_CHNLERRSTS_GET);
   65: XIC(DO3_CHNLERRSTS_TRG_GET)MSG(DO3_CHNLERRSTS_GET);
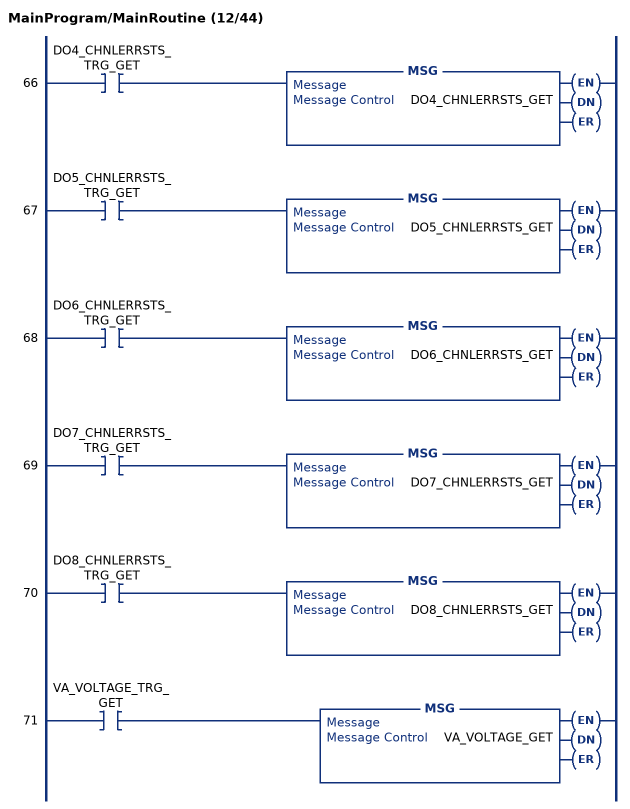
   66: XIC(DO4_CHNLERRSTS_TRG_GET)MSG(DO4_CHNLERRSTS_GET);
   67: XIC(DO5_CHNLERRSTS_TRG_GET)MSG(DO5_CHNLERRSTS_GET);
   68: XIC(DO6_CHNLERRSTS_TRG_GET)MSG(DO6_CHNLERRSTS_GET);
   69: XIC(DO7_CHNLERRSTS_TRG_GET)MSG(DO7_CHNLERRSTS_GET);
   70: XIC(DO8_CHNLERRSTS_TRG_GET)MSG(DO8_CHNLERRSTS_GET);
   71: XIC(VA_VOLTAGE_TRG_GET)MSG(VA_VOLTAGE_GET);
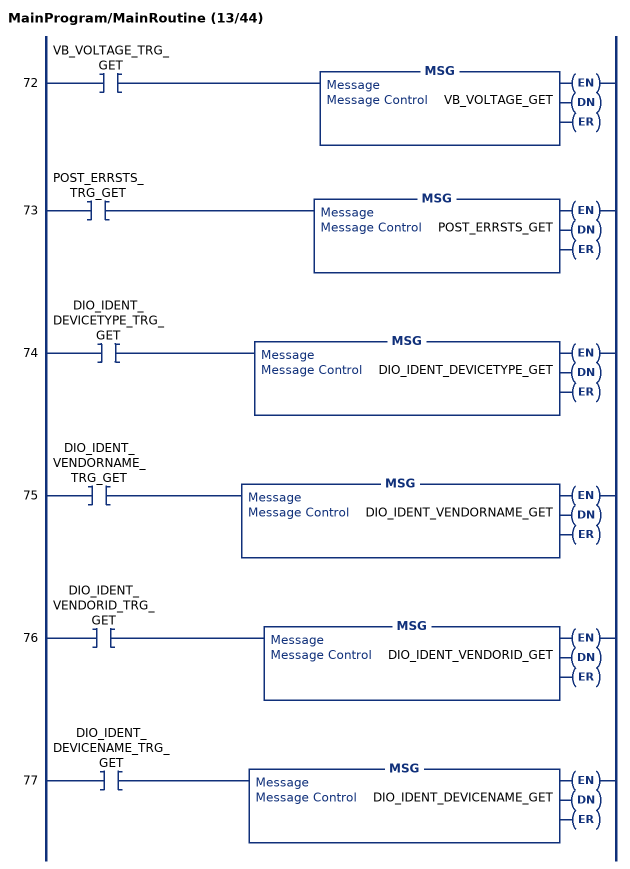
   72: XIC(VB_VOLTAGE_TRG_GET)MSG(VB_VOLTAGE_GET);
   73: XIC(POST_ERRSTS_TRG_GET)MSG(POST_ERRSTS_GET);
   74: XIC(DIO_IDENT_DEVICETYPE_TRG_GET)MSG(DIO_IDENT_DEVICETYPE_GET);
   75: XIC(DIO_IDENT_VENDORNAME_TRG_GET)MSG(DIO_IDENT_VENDORNAME_GET);
   76: XIC(DIO_IDENT_VENDORID_TRG_GET)MSG(DIO_IDENT_VENDORID_GET);
   77: XIC(DIO_IDENT_DEVICENAME_TRG_GET)MSG(DIO_IDENT_DEVICENAME_GET);
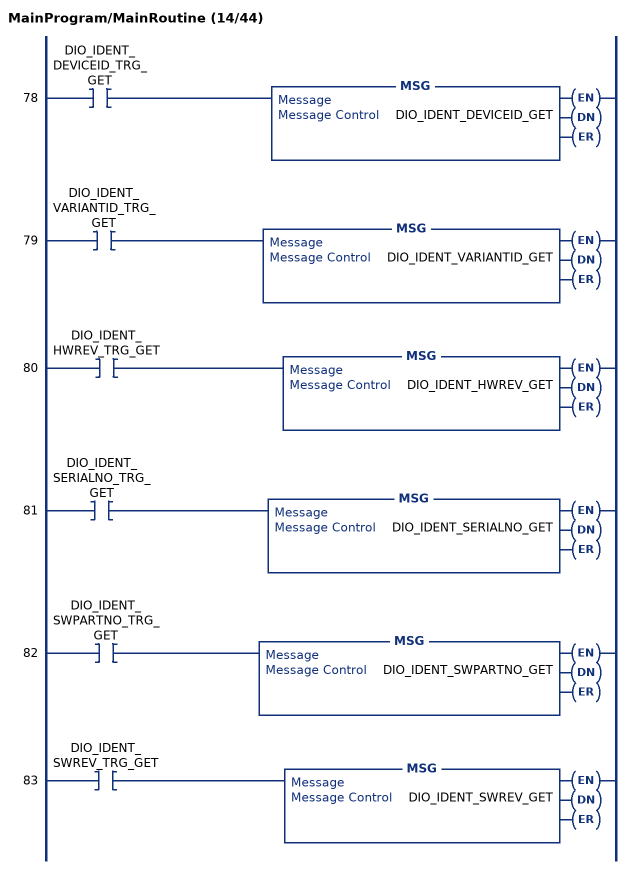
   78: XIC(DIO_IDENT_DEVICEID_TRG_GET)MSG(DIO_IDENT_DEVICEID_GET);
   79: XIC(DIO_IDENT_VARIANTID_TRG_GET)MSG(DIO_IDENT_VARIANTID_GET);
   80: XIC(DIO_IDENT_HWREV_TRG_GET)MSG(DIO_IDENT_HWREV_GET);
   81: XIC(DIO_IDENT_SERIALNO_TRG_GET)MSG(DIO_IDENT_SERIALNO_GET);
   82: XIC(DIO_IDENT_SWPARTNO_TRG_GET)MSG(DIO_IDENT_SWPARTNO_GET);
   83: XIC(DIO_IDENT_SWREV_TRG_GET)MSG(DIO_IDENT_SWREV_GET);
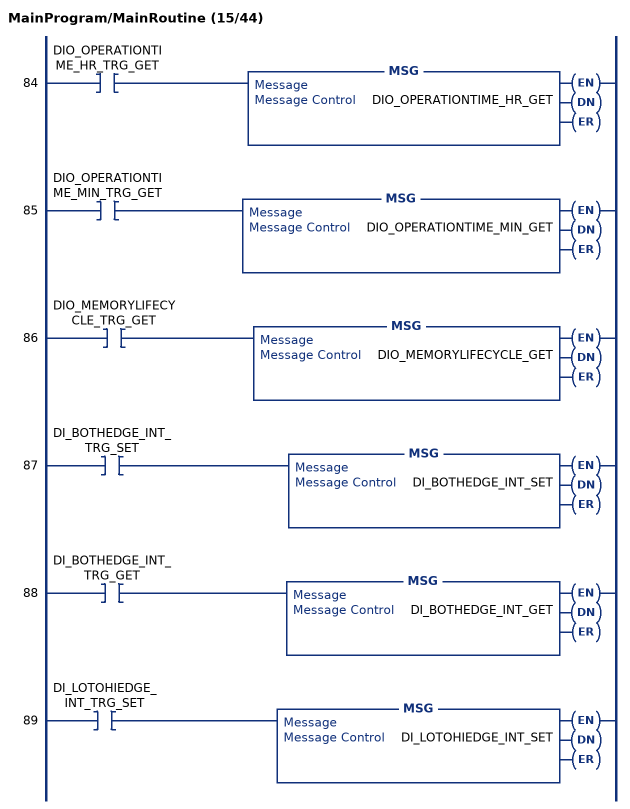
   84: XIC(DIO_OPERATIONTIME_HR_TRG_GET)MSG(DIO_OPERATIONTIME_HR_GET);
   85: XIC(DIO_OPERATIONTIME_MIN_TRG_GET)MSG(DIO_OPERATIONTIME_MIN_GET);
   86: XIC(DIO_MEMORYLIFECYCLE_TRG_GET)MSG(DIO_MEMORYLIFECYCLE_GET);
   87: XIC(DI_BOTHEDGE_INT_TRG_SET)MSG(DI_BOTHEDGE_INT_SET);
   88: XIC(DI_BOTHEDGE_INT_TRG_GET)MSG(DI_BOTHEDGE_INT_GET);
   89: XIC(DI_LOTOHIEDGE_INT_TRG_SET)MSG(DI_LOTOHIEDGE_INT_SET);
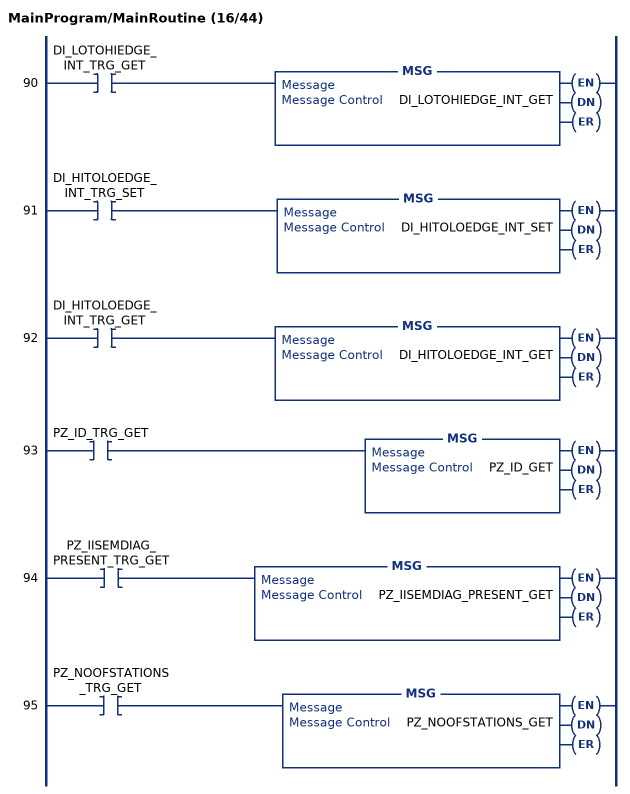
   90: XIC(DI_LOTOHIEDGE_INT_TRG_GET)MSG(DI_LOTOHIEDGE_INT_GET);
   91: XIC(DI_HITOLOEDGE_INT_TRG_SET)MSG(DI_HITOLOEDGE_INT_SET);
   92: XIC(DI_HITOLOEDGE_INT_TRG_GET)MSG(DI_HITOLOEDGE_INT_GET);
   93: XIC(PZ_ID_TRG_GET)MSG(PZ_ID_GET);
   94: XIC(PZ_IISEMDIAG_PRESENT_TRG_GET)MSG(PZ_IISEMDIAG_PRESENT_GET);
   95: XIC(PZ_NOOFSTATIONS_TRG_GET)MSG(PZ_NOOFSTATIONS_GET);
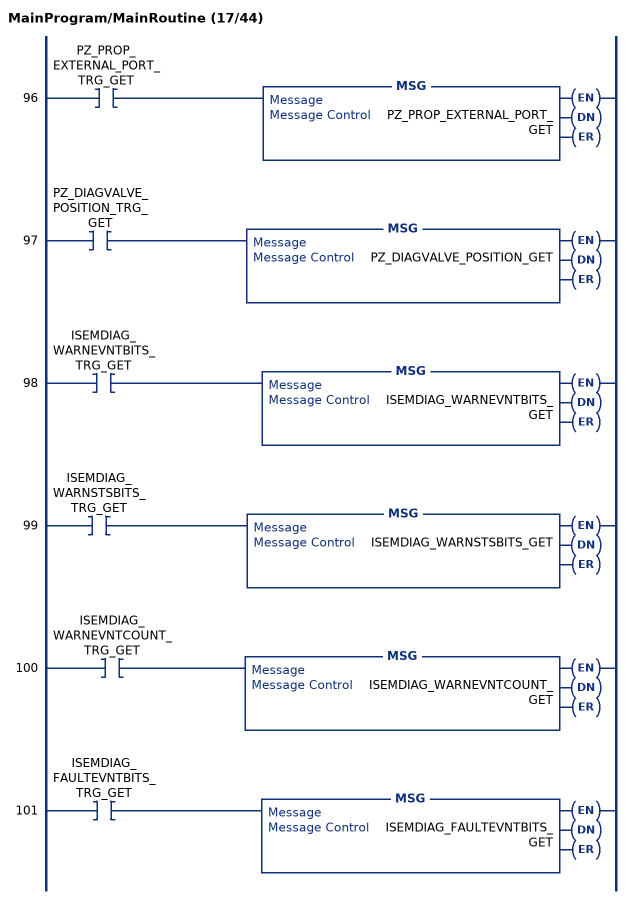
   96: XIC(PZ_PROP_EXTERNAL_PORT_TRG_GET)MSG(PZ_PROP_EXTERNAL_PORT_GET);
   97: XIC(PZ_DIAGVALVE_POSITION_TRG_GET)MSG(PZ_DIAGVALVE_POSITION_GET);
   98: XIC(ISEMDIAG_WARNEVNTBITS_TRG_GET)MSG(ISEMDIAG_WARNEVNTBITS_GET);
   99: XIC(ISEMDIAG_WARNSTSBITS_TRG_GET)MSG(ISEMDIAG_WARNSTSBITS_GET);
   100: XIC(ISEMDIAG_WARNEVNTCOUNT_TRG_GET)MSG(ISEMDIAG_WARNEVNTCOUNT_GET);
   101: XIC(ISEMDIAG_FAULTEVNTBITS_TRG_GET)MSG(ISEMDIAG_FAULTEVNTBITS_GET);
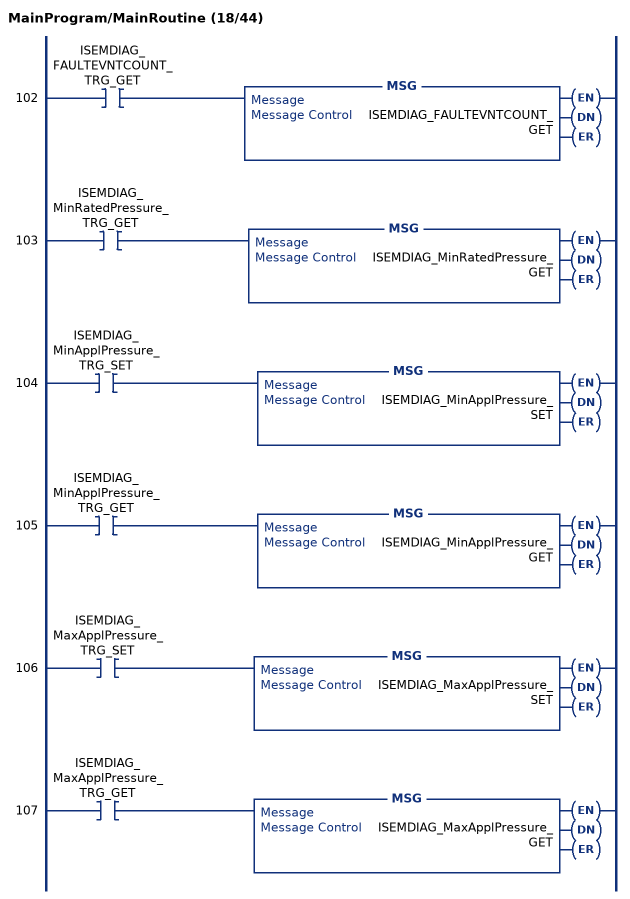
   102: XIC(ISEMDIAG_FAULTEVNTCOUNT_TRG_GET)MSG(ISEMDIAG_FAULTEVNTCOUNT_GET);
   103: XIC(ISEMDIAG_MinRatedPressure_TRG_GET)MSG(ISEMDIAG_MinRatedPressure_GET);
   104: XIC(ISEMDIAG_MinApplPressure_TRG_SET)MSG(ISEMDIAG_MinApplPressure_SET);
   105: XIC(ISEMDIAG_MinApplPressure_TRG_GET)MSG(ISEMDIAG_MinApplPressure_GET);
   106: XIC(ISEMDIAG_MaxApplPressure_TRG_SET)MSG(ISEMDIAG_MaxApplPressure_SET);
   107: XIC(ISEMDIAG_MaxApplPressure_TRG_GET)MSG(ISEMDIAG_MaxApplPressure_GET);
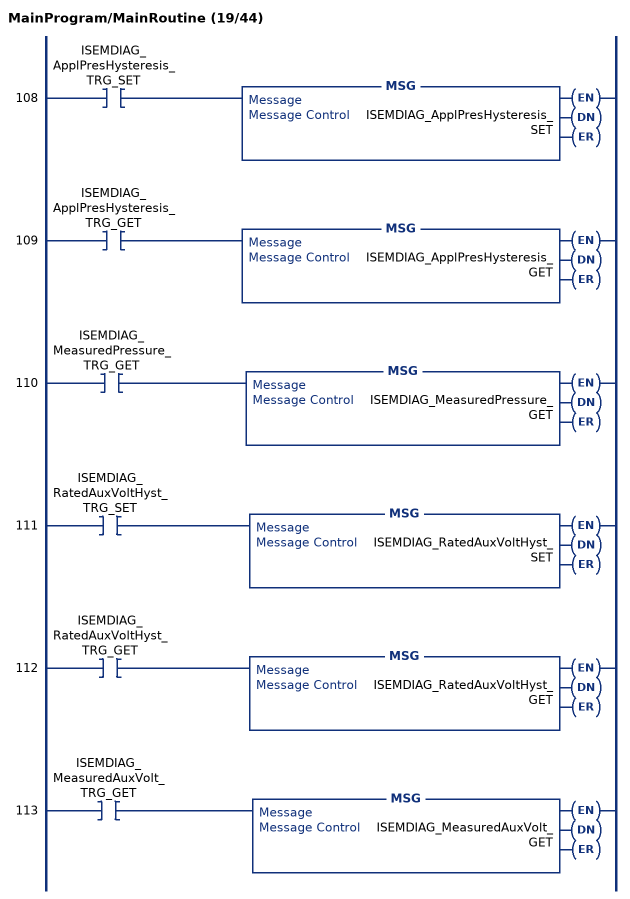
   108: XIC(ISEMDIAG_ApplPresHysteresis_TRG_SET)MSG(ISEMDIAG_ApplPresHysteresis_SET);
   109: XIC(ISEMDIAG_ApplPresHysteresis_TRG_GET)MSG(ISEMDIAG_ApplPresHysteresis_GET);
   110: XIC(ISEMDIAG_MeasuredPressure_TRG_GET)MSG(ISEMDIAG_MeasuredPressure_GET);
   111: XIC(ISEMDIAG_RatedAuxVoltHyst_TRG_SET)MSG(ISEMDIAG_RatedAuxVoltHyst_SET);
   112: XIC(ISEMDIAG_RatedAuxVoltHyst_TRG_GET)MSG(ISEMDIAG_RatedAuxVoltHyst_GET);
   113: XIC(ISEMDIAG_MeasuredAuxVolt_TRG_GET)MSG(ISEMDIAG_MeasuredAuxVolt_GET);
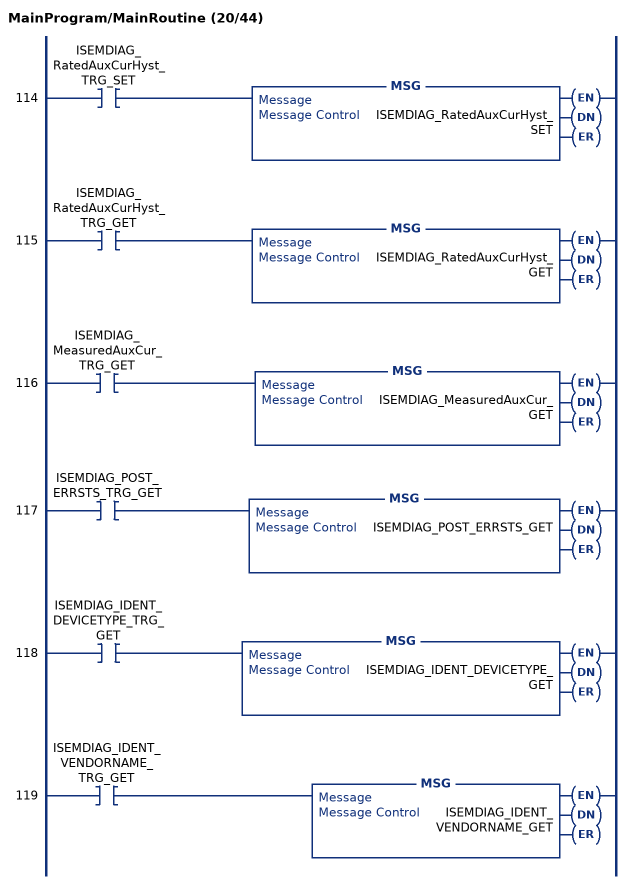
   114: XIC(ISEMDIAG_RatedAuxCurHyst_TRG_SET)MSG(ISEMDIAG_RatedAuxCurHyst_SET);
   115: XIC(ISEMDIAG_RatedAuxCurHyst_TRG_GET)MSG(ISEMDIAG_RatedAuxCurHyst_GET);
   116: XIC(ISEMDIAG_MeasuredAuxCur_TRG_GET)MSG(ISEMDIAG_MeasuredAuxCur_GET);
   117: XIC(ISEMDIAG_POST_ERRSTS_TRG_GET)MSG(ISEMDIAG_POST_ERRSTS_GET);
   118: XIC(ISEMDIAG_IDENT_DEVICETYPE_TRG_GET)MSG(ISEMDIAG_IDENT_DEVICETYPE_GET);
   119: XIC(ISEMDIAG_IDENT_VENDORNAME_TRG_GET)MSG(ISEMDIAG_IDENT_VENDORNAME_GET);
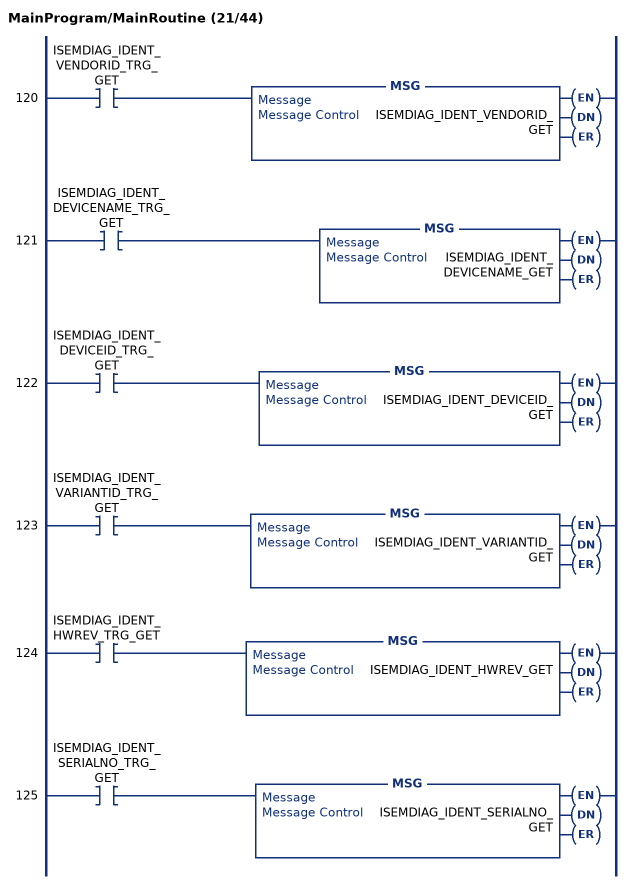
   120: XIC(ISEMDIAG_IDENT_VENDORID_TRG_GET)MSG(ISEMDIAG_IDENT_VENDORID_GET);
   121: XIC(ISEMDIAG_IDENT_DEVICENAME_TRG_GET)MSG(ISEMDIAG_IDENT_DEVICENAME_GET);
   122: XIC(ISEMDIAG_IDENT_DEVICEID_TRG_GET)MSG(ISEMDIAG_IDENT_DEVICEID_GET);
   123: XIC(ISEMDIAG_IDENT_VARIANTID_TRG_GET)MSG(ISEMDIAG_IDENT_VARIANTID_GET);
   124: XIC(ISEMDIAG_IDENT_HWREV_TRG_GET)MSG(ISEMDIAG_IDENT_HWREV_GET);
   125: XIC(ISEMDIAG_IDENT_SERIALNO_TRG_GET)MSG(ISEMDIAG_IDENT_SERIALNO_GET);
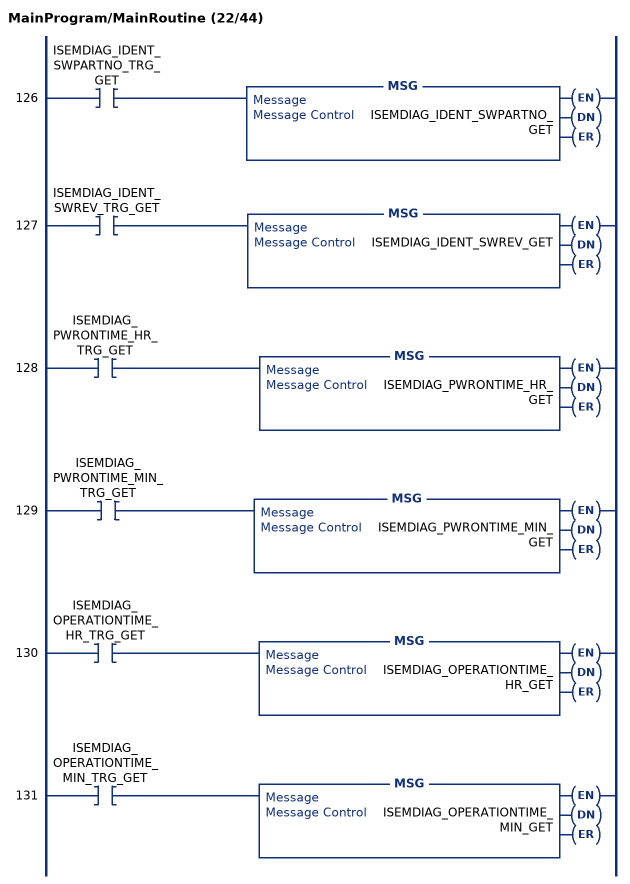
   126: XIC(ISEMDIAG_IDENT_SWPARTNO_TRG_GET)MSG(ISEMDIAG_IDENT_SWPARTNO_GET);
   127: XIC(ISEMDIAG_IDENT_SWREV_TRG_GET)MSG(ISEMDIAG_IDENT_SWREV_GET);
   128: XIC(ISEMDIAG_PWRONTIME_HR_TRG_GET)MSG(ISEMDIAG_PWRONTIME_HR_GET);
   129: XIC(ISEMDIAG_PWRONTIME_MIN_TRG_GET)MSG(ISEMDIAG_PWRONTIME_MIN_GET);
   130: XIC(ISEMDIAG_OPERATIONTIME_HR_TRG_GET)MSG(ISEMDIAG_OPERATIONTIME_HR_GET);
   131: XIC(ISEMDIAG_OPERATIONTIME_MIN_TRG_GET)MSG(ISEMDIAG_OPERATIONTIME_MIN_GET);
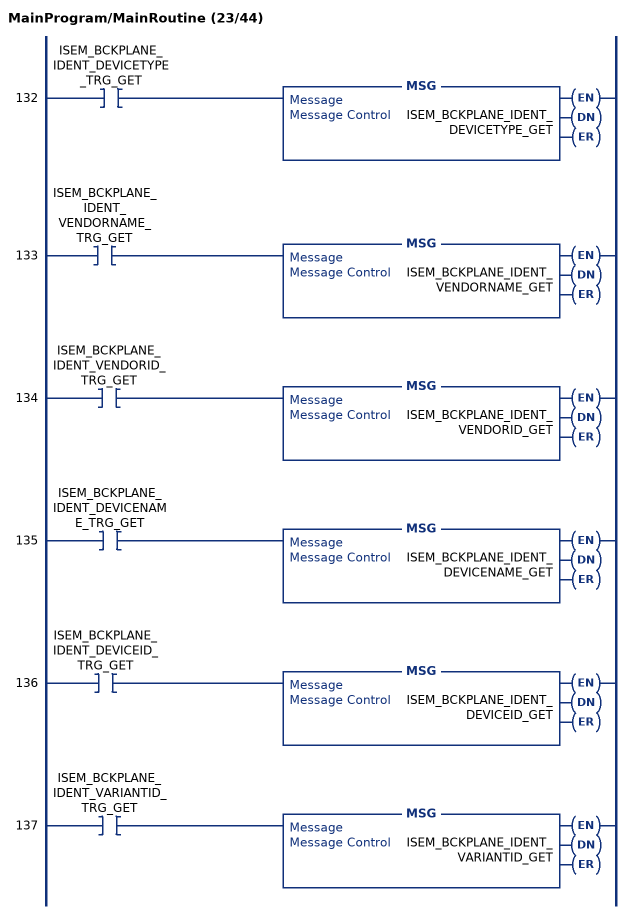
   132: XIC(ISEM_BCKPLANE_IDENT_DEVICETYPE_TRG_GET)MSG(ISEM_BCKPLANE_IDENT_DEVICETYPE_GET);
   133: XIC(ISEM_BCKPLANE_IDENT_VENDORNAME_TRG_GET)MSG(ISEM_BCKPLANE_IDENT_VENDORNAME_GET);
   134: XIC(ISEM_BCKPLANE_IDENT_VENDORID_TRG_GET)MSG(ISEM_BCKPLANE_IDENT_VENDORID_GET);
   135: XIC(ISEM_BCKPLANE_IDENT_DEVICENAME_TRG_GET)MSG(ISEM_BCKPLANE_IDENT_DEVICENAME_GET);
   136: XIC(ISEM_BCKPLANE_IDENT_DEVICEID_TRG_GET)MSG(ISEM_BCKPLANE_IDENT_DEVICEID_GET);
   137: XIC(ISEM_BCKPLANE_IDENT_VARIANTID_TRG_GET)MSG(ISEM_BCKPLANE_IDENT_VARIANTID_GET);
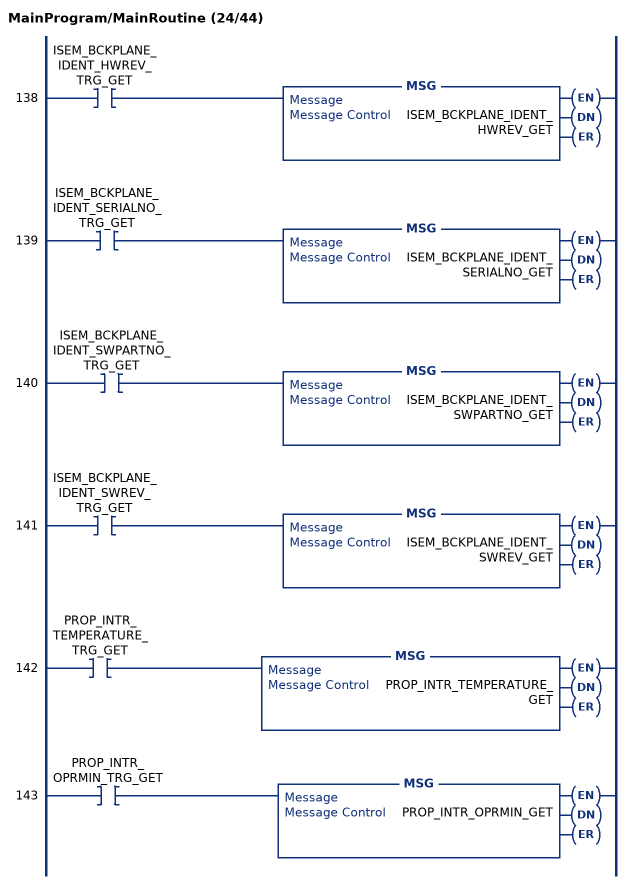
   138: XIC(ISEM_BCKPLANE_IDENT_HWREV_TRG_GET)MSG(ISEM_BCKPLANE_IDENT_HWREV_GET);
   139: XIC(ISEM_BCKPLANE_IDENT_SERIALNO_TRG_GET)MSG(ISEM_BCKPLANE_IDENT_SERIALNO_GET);
   140: XIC(ISEM_BCKPLANE_IDENT_SWPARTNO_TRG_GET)MSG(ISEM_BCKPLANE_IDENT_SWPARTNO_GET);
   141: XIC(ISEM_BCKPLANE_IDENT_SWREV_TRG_GET)MSG(ISEM_BCKPLANE_IDENT_SWREV_GET);
   142: XIC(PROP_INTR_TEMPERATURE_TRG_GET)MSG(PROP_INTR_TEMPERATURE_GET);
   143: XIC(PROP_INTR_OPRMIN_TRG_GET)MSG(PROP_INTR_OPRMIN_GET);
